Yaskawa INFORM job: A_ROOF_UPPER_0614_2_PAINT_15.JBI

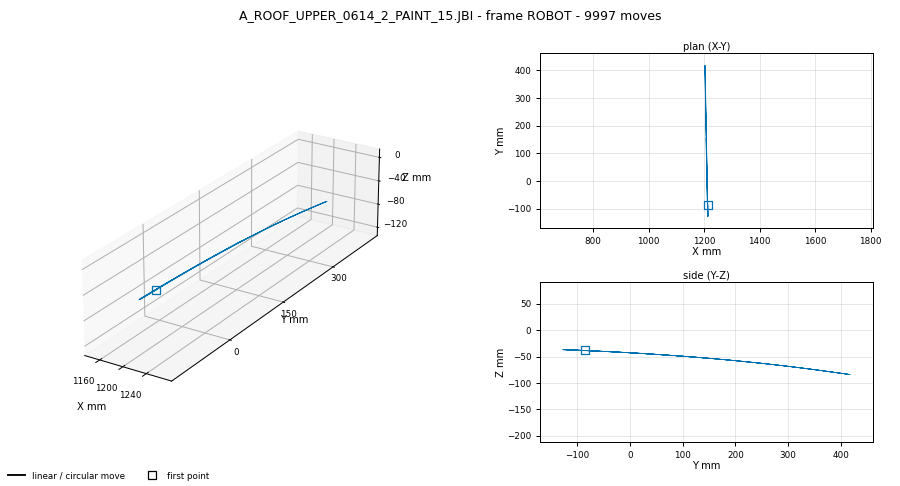
[picture p0: tool path of A_ROOF_UPPER_0614_2_PAINT_15.JBI in frame ROBOT, 9997 of 9997 moves have a stored position in this frame; points joined in program order, loops and branches not executed]
/JOB
//NAME A_ROOF_UPPER_0614_2_PAINT15
//POS
///NPOS 9997,0,0,0,0,0
///TOOL 1
///USER 0
///POSTYPE ROBOT
///RECTAN
///RCONF 1,0,0,0,0,0,0,0,0,0,0,0,0,0,0,0,0,0,0,0,0,0,0,0
C00000=1213.406,-85.221,-38.289,179.521,5.425,149.092
C00001=1213.411,-85.470,-38.278,179.518,5.424,149.093
C00002=1213.416,-85.720,-38.268,179.516,5.425,149.094
C00003=1213.422,-85.969,-38.257,179.513,5.424,149.094
C00004=1213.427,-86.220,-38.246,179.511,5.425,149.095
C00005=1213.432,-86.469,-38.234,179.509,5.424,149.095
C00006=1213.438,-86.719,-38.224,179.507,5.424,149.096
C00007=1213.443,-86.969,-38.213,179.504,5.424,149.097
C00008=1213.448,-87.218,-38.203,179.502,5.423,149.098
C00009=1213.453,-87.468,-38.192,179.500,5.424,149.098
C00010=1213.458,-87.717,-38.181,179.497,5.423,149.099
C00011=1213.463,-87.968,-38.170,179.495,5.424,149.100
C00012=1213.469,-88.217,-38.160,179.493,5.423,149.100
C00013=1213.474,-88.467,-38.149,179.491,5.423,149.101
C00014=1213.479,-88.717,-38.138,179.488,5.423,149.102
C00015=1213.484,-88.967,-38.128,179.486,5.423,149.102
C00016=1213.489,-89.216,-38.117,179.483,5.423,149.103
C00017=1213.495,-89.466,-38.107,179.481,5.423,149.104
C00018=1213.500,-89.716,-38.096,179.478,5.423,149.105
C00019=1213.506,-89.965,-38.085,179.477,5.423,149.105
C00020=1213.511,-90.215,-38.074,179.474,5.422,149.106
C00021=1213.516,-90.465,-38.064,179.472,5.423,149.106
C00022=1213.521,-90.715,-38.053,179.469,5.422,149.107
C00023=1213.526,-90.964,-38.042,179.467,5.423,149.108
C00024=1213.531,-91.214,-38.032,179.465,5.422,149.109
C00025=1213.537,-91.463,-38.021,179.463,5.422,149.109
C00026=1213.542,-91.714,-38.010,179.460,5.422,149.110
C00027=1213.547,-91.963,-38.000,179.458,5.421,149.110
C00028=1213.552,-92.213,-37.989,179.456,5.422,149.111
C00029=1213.558,-92.462,-37.979,179.453,5.421,149.112
C00030=1213.563,-92.713,-37.968,179.451,5.422,149.113
C00031=1213.568,-92.962,-37.958,179.449,5.421,149.113
C00032=1213.573,-93.212,-37.947,179.446,5.421,149.114
C00033=1213.578,-93.461,-37.936,179.444,5.421,149.114
C00034=1213.584,-93.711,-37.926,179.442,5.421,149.115
C00035=1213.589,-93.961,-37.915,179.439,5.421,149.116
C00036=1213.595,-94.211,-37.905,179.437,5.421,149.117
C00037=1213.599,-94.460,-37.894,179.435,5.420,149.117
C00038=1213.605,-94.710,-37.884,179.433,5.421,149.118
C00039=1213.610,-94.960,-37.873,179.430,5.420,149.119
C00040=1213.615,-95.209,-37.864,179.428,5.421,149.119
C00041=1213.620,-95.459,-37.853,179.425,5.420,149.120
C00042=1213.625,-95.709,-37.843,179.423,5.421,149.121
C00043=1213.631,-95.958,-37.832,179.421,5.420,149.121
C00044=1213.636,-96.208,-37.821,179.419,5.420,149.122
C00045=1213.641,-96.458,-37.811,179.416,5.420,149.123
C00046=1213.646,-96.708,-37.801,179.414,5.420,149.123
C00047=1213.652,-96.957,-37.790,179.411,5.420,149.124
C00048=1213.657,-97.208,-37.780,179.409,5.420,149.125
C00049=1213.662,-97.457,-37.770,179.407,5.419,149.125
C00050=1213.668,-97.706,-37.759,179.405,5.420,149.126
C00051=1213.673,-97.956,-37.748,179.402,5.419,149.127
C00052=1213.678,-98.206,-37.738,179.400,5.419,149.127
C00053=1213.683,-98.456,-37.728,179.398,5.419,149.128
C00054=1213.688,-98.705,-37.718,179.396,5.419,149.129
C00055=1213.694,-98.955,-37.707,179.393,5.419,149.129
C00056=1213.699,-99.205,-37.697,179.391,5.419,149.130
C00057=1213.704,-99.455,-37.687,179.389,5.419,149.131
C00058=1213.709,-99.705,-37.676,179.387,5.419,149.131
C00059=1213.715,-99.955,-37.666,179.384,5.419,149.132
C00060=1213.720,-100.204,-37.656,179.382,5.419,149.133
C00061=1213.725,-100.454,-37.646,179.380,5.418,149.133
C00062=1213.731,-100.725,-37.635,179.377,5.418,149.134
C00063=1213.737,-100.996,-37.624,179.375,5.418,149.135
C00064=1213.743,-101.268,-37.612,179.372,5.418,149.135
C00065=1213.747,-101.539,-37.600,179.370,5.418,149.136
C00066=1213.753,-101.788,-37.590,179.367,5.418,149.137
C00067=1213.759,-102.038,-37.580,179.365,5.418,149.138
C00068=1213.763,-102.288,-37.570,179.363,5.418,149.138
C00069=1213.768,-102.537,-37.560,179.360,5.418,149.139
C00070=1213.774,-102.787,-37.550,179.358,5.417,149.139
C00071=1213.779,-103.038,-37.540,179.356,5.417,149.140
C00072=1213.785,-103.287,-37.529,179.354,5.417,149.141
C00073=1213.790,-103.536,-37.520,179.351,5.417,149.142
C00074=1213.795,-103.787,-37.509,179.349,5.417,149.142
C00075=1213.800,-104.036,-37.499,179.347,5.417,149.143
C00076=1213.806,-104.286,-37.489,179.344,5.417,149.144
C00077=1213.810,-104.536,-37.479,179.342,5.417,149.144
C00078=1213.816,-104.785,-37.469,179.340,5.417,149.145
C00079=1213.821,-105.035,-37.458,179.338,5.417,149.146
C00080=1213.826,-105.285,-37.448,179.335,5.417,149.146
C00081=1213.831,-105.534,-37.438,179.333,5.416,149.147
C00082=1213.837,-105.784,-37.428,179.331,5.416,149.148
C00083=1213.842,-106.034,-37.418,179.329,5.416,149.148
C00084=1213.848,-106.284,-37.408,179.326,5.416,149.149
C00085=1213.853,-106.533,-37.398,179.324,5.416,149.150
C00086=1213.858,-106.784,-37.388,179.322,5.416,149.150
C00087=1213.863,-107.033,-37.378,179.320,5.416,149.151
C00088=1213.868,-107.282,-37.368,179.317,5.416,149.152
C00089=1213.874,-107.532,-37.358,179.315,5.416,149.152
C00090=1213.879,-107.782,-37.347,179.313,5.415,149.153
C00091=1213.885,-108.032,-37.338,179.311,5.416,149.154
C00092=1213.890,-108.281,-37.328,179.308,5.415,149.154
C00093=1213.895,-108.532,-37.318,179.306,5.415,149.155
C00094=1213.900,-108.781,-37.307,179.303,5.415,149.156
C00095=1213.905,-109.031,-37.298,179.301,5.415,149.156
C00096=1213.911,-109.280,-37.288,179.299,5.415,149.157
C00097=1213.916,-109.531,-37.278,179.297,5.415,149.158
C00098=1213.921,-109.780,-37.268,179.295,5.415,149.158
C00099=1213.926,-110.030,-37.258,179.292,5.415,149.159
C00100=1213.932,-110.279,-37.248,179.290,5.415,149.160
C00101=1213.936,-110.530,-37.238,179.288,5.415,149.160
C00102=1213.942,-110.779,-37.228,179.286,5.415,149.161
C00103=1213.947,-111.029,-37.219,179.283,5.415,149.162
C00104=1213.953,-111.278,-37.208,179.281,5.415,149.162
C00105=1213.958,-111.528,-37.198,179.279,5.414,149.163
C00106=1213.963,-111.778,-37.189,179.277,5.415,149.164
C00107=1213.968,-112.028,-37.179,179.274,5.414,149.164
C00108=1213.974,-112.277,-37.168,179.272,5.414,149.165
C00109=1213.979,-112.527,-37.160,179.270,5.414,149.166
C00110=1213.984,-112.777,-37.149,179.267,5.414,149.166
C00111=1213.989,-113.027,-37.139,179.265,5.414,149.167
C00112=1213.995,-113.276,-37.129,179.263,5.414,149.168
C00113=1214.000,-113.526,-37.120,179.260,5.413,149.168
C00114=1214.005,-113.776,-37.110,179.258,5.414,149.169
C00115=1214.010,-114.026,-37.099,179.256,5.413,149.170
C00116=1214.015,-114.276,-37.091,179.254,5.414,149.170
C00117=1214.021,-114.525,-37.080,179.251,5.413,149.171
C00118=1214.026,-114.774,-37.071,179.249,5.413,149.171
C00119=1214.032,-115.025,-37.061,179.247,5.414,149.172
C00120=1214.037,-115.275,-37.051,179.245,5.413,149.173
C00121=1214.042,-115.525,-37.042,179.243,5.413,149.173
C00122=1214.048,-115.774,-37.032,179.240,5.413,149.174
C00123=1214.052,-116.023,-37.022,179.238,5.413,149.175
C00124=1214.058,-116.274,-37.012,179.236,5.413,149.176
C00125=1214.063,-116.523,-37.003,179.233,5.413,149.176
C00126=1214.068,-116.773,-36.992,179.231,5.412,149.177
C00127=1214.073,-117.023,-36.983,179.229,5.413,149.177
C00128=1214.079,-117.272,-36.973,179.226,5.412,149.178
C00129=1214.084,-117.522,-36.964,179.224,5.413,149.179
C00130=1214.090,-117.772,-36.954,179.222,5.412,149.179
C00131=1214.095,-118.021,-36.944,179.220,5.412,149.180
C00132=1214.100,-118.272,-36.935,179.217,5.412,149.181
C00133=1214.105,-118.521,-36.925,179.215,5.412,149.182
C00134=1214.111,-118.771,-36.915,179.213,5.411,149.182
C00135=1214.116,-119.021,-36.906,179.211,5.412,149.183
C00136=1214.121,-119.271,-36.896,179.209,5.412,149.183
C00137=1214.126,-119.520,-36.887,179.206,5.412,149.184
C00138=1214.132,-119.770,-36.877,179.205,5.412,149.185
C00139=1214.137,-120.019,-36.868,179.202,5.411,149.185
C00140=1214.142,-120.270,-36.858,179.200,5.412,149.186
C00141=1214.147,-120.520,-36.848,179.198,5.411,149.187
C00142=1214.153,-120.770,-36.839,179.196,5.411,149.187
C00143=1214.158,-121.019,-36.829,179.193,5.411,149.188
C00144=1214.163,-121.269,-36.820,179.191,5.411,149.189
C00145=1214.169,-121.518,-36.810,179.189,5.411,149.189
C00146=1214.174,-121.768,-36.801,179.187,5.411,149.190
C00147=1214.180,-122.018,-36.791,179.184,5.411,149.191
C00148=1214.185,-122.268,-36.782,179.182,5.411,149.191
C00149=1214.190,-122.518,-36.771,179.180,5.411,149.192
C00150=1214.195,-122.768,-36.762,179.178,5.411,149.193
C00151=1214.200,-123.017,-36.753,179.175,5.411,149.193
C00152=1214.206,-123.267,-36.743,179.173,5.410,149.194
C00153=1214.211,-123.517,-36.734,179.171,5.410,149.194
C00154=1214.216,-123.766,-36.724,179.168,5.410,149.195
C00155=1214.222,-124.016,-36.715,179.166,5.410,149.196
C00156=1214.226,-124.265,-36.706,179.164,5.410,149.196
C00157=1214.232,-124.516,-36.696,179.162,5.410,149.197
C00158=1214.237,-124.765,-36.687,179.159,5.410,149.198
C00159=1214.242,-125.015,-36.678,179.157,5.410,149.199
C00160=1214.248,-125.265,-36.668,179.156,5.410,149.199
C00161=1214.253,-125.514,-36.659,179.153,5.410,149.200
C00162=1214.259,-125.764,-36.649,179.151,5.410,149.200
C00163=1214.264,-126.014,-36.640,179.148,5.410,149.201
C00164=1214.268,-126.264,-36.630,179.147,5.410,149.202
C00165=1214.274,-126.514,-36.621,179.144,5.409,149.202
C00166=1213.853,-126.525,-36.659,179.140,5.412,149.204
C00167=1213.848,-126.275,-36.668,179.142,5.413,149.204
C00168=1213.842,-126.025,-36.677,179.144,5.413,149.203
C00169=1213.837,-125.775,-36.687,179.147,5.413,149.202
C00170=1213.832,-125.526,-36.696,179.149,5.413,149.202
C00171=1213.826,-125.276,-36.705,179.151,5.414,149.201
C00172=1213.821,-125.026,-36.715,179.153,5.413,149.200
C00173=1213.816,-124.776,-36.724,179.155,5.413,149.200
C00174=1213.810,-124.527,-36.734,179.158,5.414,149.199
C00175=1213.805,-124.277,-36.743,179.160,5.413,149.198
C00176=1213.800,-124.027,-36.752,179.162,5.414,149.198
C00177=1213.794,-123.777,-36.762,179.165,5.413,149.197
C00178=1213.790,-123.527,-36.771,179.167,5.414,149.197
C00179=1213.785,-123.278,-36.781,179.169,5.414,149.196
C00180=1213.779,-123.028,-36.790,179.172,5.414,149.195
C00181=1213.774,-122.778,-36.799,179.173,5.414,149.195
C00182=1213.768,-122.528,-36.809,179.176,5.414,149.194
C00183=1213.763,-122.278,-36.818,179.178,5.414,149.193
C00184=1213.758,-122.029,-36.828,179.180,5.414,149.193
C00185=1213.752,-121.779,-36.837,179.182,5.414,149.192
C00186=1213.747,-121.530,-36.847,179.184,5.414,149.191
C00187=1213.741,-121.279,-36.857,179.187,5.415,149.191
C00188=1213.737,-121.030,-36.866,179.189,5.414,149.190
C00189=1213.731,-120.779,-36.876,179.191,5.415,149.189
C00190=1213.726,-120.530,-36.886,179.193,5.415,149.189
C00191=1213.720,-120.280,-36.895,179.196,5.415,149.188
C00192=1213.716,-120.031,-36.905,179.198,5.415,149.187
C00193=1213.710,-119.781,-36.914,179.200,5.415,149.187
C00194=1213.705,-119.531,-36.924,179.202,5.415,149.186
C00195=1213.700,-119.282,-36.933,179.205,5.415,149.185
C00196=1213.694,-119.032,-36.943,179.207,5.415,149.185
C00197=1213.689,-118.782,-36.952,179.209,5.415,149.184
C00198=1213.684,-118.532,-36.962,179.211,5.415,149.183
C00199=1213.679,-118.282,-36.971,179.213,5.415,149.183
C00200=1213.673,-118.032,-36.982,179.216,5.416,149.182
C00201=1213.668,-117.783,-36.991,179.218,5.415,149.181
C00202=1213.662,-117.533,-37.001,179.220,5.416,149.181
C00203=1213.658,-117.284,-37.010,179.223,5.415,149.180
C00204=1213.652,-117.033,-37.020,179.225,5.416,149.180
C00205=1213.647,-116.784,-37.030,179.227,5.416,149.179
C00206=1213.641,-116.534,-37.039,179.230,5.416,149.178
C00207=1213.637,-116.284,-37.049,179.232,5.416,149.177
C00208=1213.631,-116.035,-37.059,179.234,5.417,149.177
C00209=1213.626,-115.785,-37.068,179.236,5.416,149.176
C00210=1213.621,-115.535,-37.079,179.239,5.417,149.175
C00211=1213.616,-115.286,-37.088,179.241,5.416,149.175
C00212=1213.610,-115.035,-37.098,179.243,5.417,149.174
C00213=1213.604,-114.786,-37.108,179.245,5.417,149.174
C00214=1213.599,-114.536,-37.117,179.247,5.416,149.173
C00215=1213.594,-114.286,-37.127,179.250,5.417,149.172
C00216=1213.589,-114.036,-37.137,179.251,5.417,149.172
C00217=1213.584,-113.786,-37.146,179.254,5.417,149.171
C00218=1213.579,-113.537,-37.156,179.256,5.417,149.170
C00219=1213.573,-113.288,-37.166,179.259,5.417,149.170
C00220=1213.567,-113.037,-37.176,179.261,5.417,149.169
C00221=1213.563,-112.787,-37.186,179.263,5.418,149.168
C00222=1213.557,-112.538,-37.196,179.265,5.417,149.168
C00223=1213.552,-112.289,-37.206,179.268,5.418,149.167
C00224=1213.547,-112.038,-37.215,179.270,5.417,149.166
C00225=1213.541,-111.789,-37.225,179.272,5.418,149.166
C00226=1213.537,-111.539,-37.235,179.274,5.418,149.165
C00227=1213.531,-111.289,-37.245,179.277,5.418,149.164
C00228=1213.525,-111.039,-37.255,179.279,5.418,149.164
C00229=1213.520,-110.790,-37.265,179.281,5.419,149.163
C00230=1213.515,-110.540,-37.275,179.283,5.418,149.162
C00231=1213.510,-110.291,-37.285,179.286,5.419,149.162
C00232=1213.505,-110.040,-37.294,179.288,5.418,149.161
C00233=1213.499,-109.791,-37.304,179.291,5.419,149.160
C00234=1213.495,-109.541,-37.314,179.292,5.419,149.160
C00235=1213.489,-109.291,-37.325,179.294,5.418,149.159
C00236=1213.483,-109.041,-37.334,179.297,5.419,149.158
C00237=1213.478,-108.792,-37.344,179.299,5.418,149.158
C00238=1213.473,-108.542,-37.354,179.302,5.419,149.157
C00239=1213.468,-108.292,-37.364,179.303,5.419,149.156
C00240=1213.463,-108.043,-37.374,179.306,5.419,149.156
C00241=1213.457,-107.793,-37.384,179.308,5.419,149.155
C00242=1213.452,-107.543,-37.394,179.311,5.419,149.154
C00243=1213.446,-107.293,-37.404,179.312,5.419,149.154
C00244=1213.442,-107.044,-37.414,179.315,5.420,149.153
C00245=1213.437,-106.794,-37.425,179.317,5.419,149.152
C00246=1213.431,-106.544,-37.435,179.320,5.420,149.152
C00247=1213.426,-106.295,-37.444,179.322,5.419,149.151
C00248=1213.420,-106.045,-37.455,179.324,5.420,149.150
C00249=1213.415,-105.794,-37.464,179.326,5.420,149.150
C00250=1213.410,-105.545,-37.475,179.329,5.420,149.149
C00251=1213.405,-105.296,-37.484,179.331,5.420,149.148
C00252=1213.400,-105.045,-37.495,179.334,5.420,149.148
C00253=1213.394,-104.796,-37.505,179.335,5.420,149.147
C00254=1213.389,-104.546,-37.515,179.338,5.420,149.146
C00255=1213.384,-104.296,-37.525,179.340,5.420,149.146
C00256=1213.379,-104.047,-37.535,179.343,5.421,149.145
C00257=1213.373,-103.797,-37.546,179.345,5.420,149.144
C00258=1213.368,-103.547,-37.556,179.347,5.421,149.144
C00259=1213.363,-103.298,-37.566,179.349,5.421,149.143
C00260=1213.358,-103.048,-37.576,179.352,5.421,149.142
C00261=1213.353,-102.798,-37.587,179.354,5.421,149.142
C00262=1213.347,-102.548,-37.597,179.357,5.421,149.141
C00263=1213.342,-102.299,-37.606,179.358,5.421,149.140
C00264=1213.337,-102.049,-37.617,179.361,5.421,149.140
C00265=1213.332,-101.799,-37.627,179.363,5.421,149.139
C00266=1213.326,-101.550,-37.637,179.366,5.422,149.138
C00267=1213.321,-101.279,-37.648,179.368,5.421,149.138
C00268=1213.315,-101.007,-37.660,179.370,5.422,149.137
C00269=1213.310,-100.736,-37.671,179.373,5.422,149.136
C00270=1213.303,-100.465,-37.682,179.375,5.422,149.135
C00271=1213.299,-100.215,-37.692,179.378,5.422,149.135
C00272=1213.293,-99.965,-37.702,179.380,5.422,149.134
C00273=1213.288,-99.716,-37.712,179.382,5.422,149.133
C00274=1213.283,-99.466,-37.723,179.384,5.422,149.133
C00275=1213.277,-99.216,-37.733,179.387,5.423,149.132
C00276=1213.272,-98.966,-37.744,179.389,5.422,149.131
C00277=1213.266,-98.716,-37.754,179.392,5.423,149.131
C00278=1213.262,-98.467,-37.764,179.393,5.423,149.130
C00279=1213.257,-98.217,-37.774,179.396,5.423,149.129
C00280=1213.251,-97.967,-37.784,179.398,5.423,149.129
C00281=1213.246,-97.717,-37.795,179.401,5.423,149.128
C00282=1213.241,-97.468,-37.806,179.403,5.423,149.127
C00283=1213.235,-97.218,-37.816,179.405,5.423,149.127
C00284=1213.230,-96.968,-37.827,179.407,5.423,149.126
C00285=1213.225,-96.719,-37.837,179.410,5.424,149.125
C00286=1213.220,-96.468,-37.847,179.412,5.423,149.125
C00287=1213.214,-96.219,-37.858,179.414,5.424,149.124
C00288=1213.210,-95.969,-37.868,179.417,5.423,149.123
C00289=1213.204,-95.719,-37.878,179.419,5.424,149.123
C00290=1213.199,-95.470,-37.889,179.421,5.424,149.122
C00291=1213.194,-95.220,-37.899,179.423,5.424,149.121
C00292=1213.188,-94.971,-37.910,179.426,5.424,149.121
C00293=1213.183,-94.720,-37.920,179.428,5.424,149.120
C00294=1213.178,-94.471,-37.930,179.430,5.424,149.119
C00295=1213.173,-94.221,-37.942,179.433,5.425,149.119
C00296=1213.167,-93.972,-37.952,179.435,5.424,149.118
C00297=1213.162,-93.721,-37.962,179.437,5.425,149.117
C00298=1213.157,-93.472,-37.973,179.439,5.424,149.117
C00299=1213.151,-93.222,-37.983,179.442,5.425,149.116
C00300=1213.146,-92.973,-37.994,179.444,5.424,149.115
C00301=1213.141,-92.723,-38.004,179.446,5.425,149.115
C00302=1213.136,-92.473,-38.015,179.449,5.426,149.114
C00303=1213.130,-92.223,-38.025,179.451,5.425,149.113
C00304=1213.126,-91.974,-38.036,179.454,5.426,149.113
C00305=1213.120,-91.724,-38.047,179.456,5.425,149.112
C00306=1213.115,-91.474,-38.057,179.459,5.426,149.111
C00307=1213.109,-91.224,-38.067,179.460,5.426,149.111
C00308=1213.105,-90.975,-38.079,179.463,5.426,149.110
C00309=1213.099,-90.725,-38.089,179.465,5.426,149.109
C00310=1213.094,-90.475,-38.099,179.468,5.426,149.109
C00311=1213.089,-90.226,-38.110,179.470,5.426,149.108
C00312=1213.084,-89.976,-38.121,179.472,5.426,149.107
C00313=1213.078,-89.726,-38.131,179.474,5.426,149.106
C00314=1213.073,-89.477,-38.142,179.477,5.427,149.106
C00315=1213.068,-89.227,-38.153,179.479,5.426,149.105
C00316=1213.063,-88.977,-38.163,179.481,5.427,149.104
C00317=1213.058,-88.728,-38.174,179.483,5.426,149.104
C00318=1213.053,-88.478,-38.185,179.486,5.427,149.103
C00319=1213.047,-88.228,-38.195,179.488,5.426,149.102
C00320=1213.042,-87.978,-38.207,179.490,5.427,149.102
C00321=1213.037,-87.728,-38.217,179.492,5.427,149.101
C00322=1213.031,-87.479,-38.228,179.495,5.427,149.100
C00323=1213.026,-87.229,-38.239,179.498,5.428,149.100
C00324=1213.021,-86.979,-38.249,179.500,5.427,149.099
C00325=1213.016,-86.730,-38.260,179.503,5.428,149.098
C00326=1213.010,-86.480,-38.271,179.505,5.427,149.098
C00327=1213.005,-86.230,-38.281,179.507,5.428,149.097
C00328=1213.000,-85.981,-38.292,179.509,5.428,149.096
C00329=1212.995,-85.731,-38.303,179.512,5.428,149.096
C00330=1212.990,-85.481,-38.315,179.514,5.428,149.095
C00331=1212.984,-85.231,-38.325,179.516,5.428,149.094
C00332=1212.979,-84.982,-38.336,179.518,5.428,149.094
C00333=1212.974,-84.732,-38.346,179.521,5.428,149.093
C00334=1212.969,-84.483,-38.358,179.523,5.429,149.092
C00335=1212.964,-84.232,-38.368,179.525,5.429,149.092
C00336=1212.959,-83.983,-38.379,179.527,5.429,149.091
C00337=1212.953,-83.733,-38.390,179.530,5.429,149.090
C00338=1212.947,-83.483,-38.400,179.533,5.429,149.090
C00339=1212.943,-83.234,-38.412,179.535,5.429,149.089
C00340=1212.938,-82.983,-38.422,179.538,5.430,149.088
C00341=1212.932,-82.734,-38.433,179.539,5.430,149.088
C00342=1212.928,-82.485,-38.445,179.542,5.430,149.087
C00343=1212.921,-82.235,-38.455,179.544,5.430,149.086
C00344=1212.917,-81.985,-38.467,179.547,5.430,149.086
C00345=1212.912,-81.735,-38.477,179.549,5.430,149.085
C00346=1212.906,-81.486,-38.488,179.551,5.430,149.084
C00347=1212.901,-81.236,-38.499,179.553,5.430,149.083
C00348=1212.895,-80.987,-38.510,179.556,5.431,149.083
C00349=1212.890,-80.736,-38.521,179.558,5.431,149.082
C00350=1212.886,-80.487,-38.532,179.560,5.431,149.081
C00351=1212.880,-80.238,-38.543,179.563,5.431,149.081
C00352=1212.875,-79.988,-38.554,179.565,5.431,149.080
C00353=1212.870,-79.738,-38.565,179.568,5.431,149.079
C00354=1212.864,-79.488,-38.576,179.570,5.431,149.079
C00355=1212.860,-79.239,-38.587,179.572,5.432,149.078
C00356=1212.855,-78.989,-38.598,179.574,5.431,149.077
C00357=1212.849,-78.739,-38.609,179.577,5.432,149.077
C00358=1212.844,-78.489,-38.620,179.579,5.431,149.076
C00359=1212.839,-78.239,-38.631,179.582,5.432,149.075
C00360=1212.833,-77.990,-38.642,179.584,5.432,149.075
C00361=1212.828,-77.740,-38.654,179.586,5.432,149.074
C00362=1212.823,-77.490,-38.664,179.589,5.432,149.073
C00363=1212.818,-77.241,-38.675,179.591,5.432,149.073
C00364=1212.813,-76.991,-38.687,179.593,5.433,149.072
C00365=1212.808,-76.741,-38.698,179.595,5.432,149.071
C00366=1212.802,-76.492,-38.709,179.598,5.433,149.071
C00367=1212.797,-76.242,-38.721,179.600,5.432,149.070
C00368=1212.792,-75.992,-38.731,179.603,5.433,149.069
C00369=1212.787,-75.743,-38.742,179.606,5.433,149.068
C00370=1212.781,-75.493,-38.754,179.608,5.433,149.068
C00371=1212.776,-75.222,-38.766,179.610,5.433,149.067
C00372=1212.770,-74.952,-38.777,179.613,5.434,149.066
C00373=1212.764,-74.681,-38.790,179.615,5.434,149.066
C00374=1212.759,-74.411,-38.803,179.618,5.434,149.065
C00375=1212.754,-74.161,-38.813,179.620,5.434,149.064
C00376=1212.748,-73.911,-38.825,179.622,5.434,149.064
C00377=1212.743,-73.662,-38.836,179.625,5.435,149.063
C00378=1212.739,-73.412,-38.847,179.627,5.434,149.062
C00379=1212.732,-73.162,-38.858,179.629,5.435,149.062
C00380=1212.728,-72.913,-38.869,179.631,5.435,149.061
C00381=1212.722,-72.663,-38.881,179.634,5.435,149.060
C00382=1212.717,-72.414,-38.892,179.636,5.435,149.059
C00383=1212.712,-72.164,-38.904,179.639,5.435,149.059
C00384=1212.707,-71.913,-38.915,179.642,5.436,149.058
C00385=1212.702,-71.664,-38.926,179.644,5.435,149.057
C00386=1212.696,-71.415,-38.937,179.646,5.436,149.057
C00387=1212.691,-71.165,-38.949,179.648,5.436,149.056
C00388=1212.686,-70.915,-38.960,179.651,5.436,149.055
C00389=1212.681,-70.665,-38.972,179.653,5.436,149.055
C00390=1212.675,-70.416,-38.982,179.655,5.436,149.054
C00391=1212.670,-70.166,-38.994,179.658,5.437,149.053
C00392=1212.665,-69.916,-39.005,179.660,5.436,149.053
C00393=1212.660,-69.666,-39.017,179.663,5.437,149.052
C00394=1212.655,-69.417,-39.029,179.665,5.436,149.051
C00395=1212.649,-69.168,-39.040,179.668,5.437,149.051
C00396=1212.644,-68.918,-39.051,179.669,5.437,149.050
C00397=1212.639,-68.668,-39.063,179.672,5.437,149.049
C00398=1212.634,-68.418,-39.075,179.674,5.438,149.049
C00399=1212.629,-68.168,-39.085,179.677,5.437,149.048
C00400=1212.623,-67.919,-39.097,179.679,5.438,149.047
C00401=1212.619,-67.669,-39.108,179.681,5.438,149.047
C00402=1212.613,-67.419,-39.120,179.684,5.438,149.046
C00403=1212.608,-67.170,-39.131,179.687,5.438,149.045
C00404=1212.603,-66.920,-39.143,179.689,5.438,149.044
C00405=1212.598,-66.671,-39.154,179.691,5.439,149.044
C00406=1212.592,-66.421,-39.166,179.693,5.439,149.043
C00407=1212.588,-66.171,-39.177,179.696,5.439,149.042
C00408=1212.582,-65.921,-39.189,179.698,5.439,149.042
C00409=1212.577,-65.671,-39.201,179.700,5.439,149.041
C00410=1212.572,-65.422,-39.212,179.703,5.440,149.040
C00411=1212.566,-65.173,-39.224,179.705,5.439,149.040
C00412=1212.561,-64.923,-39.235,179.708,5.440,149.039
C00413=1212.556,-64.673,-39.247,179.710,5.439,149.038
C00414=1212.551,-64.423,-39.258,179.712,5.440,149.038
C00415=1212.546,-64.173,-39.270,179.715,5.441,149.037
C00416=1212.541,-63.924,-39.281,179.717,5.440,149.036
C00417=1212.536,-63.674,-39.293,179.720,5.441,149.036
C00418=1212.530,-63.425,-39.304,179.722,5.440,149.035
C00419=1212.525,-63.175,-39.316,179.724,5.441,149.034
C00420=1212.520,-62.925,-39.328,179.727,5.441,149.034
C00421=1212.515,-62.675,-39.339,179.729,5.441,149.033
C00422=1212.510,-62.426,-39.352,179.732,5.441,149.032
C00423=1212.505,-62.176,-39.363,179.734,5.441,149.031
C00424=1212.500,-61.927,-39.375,179.736,5.442,149.031
C00425=1212.494,-61.677,-39.387,179.739,5.442,149.030
C00426=1212.489,-61.427,-39.398,179.741,5.442,149.030
C00427=1212.483,-61.178,-39.410,179.743,5.442,149.029
C00428=1212.479,-60.928,-39.421,179.745,5.442,149.028
C00429=1212.473,-60.678,-39.433,179.748,5.442,149.027
C00430=1212.468,-60.429,-39.445,179.751,5.443,149.027
C00431=1212.464,-60.179,-39.457,179.753,5.443,149.026
C00432=1212.458,-59.929,-39.469,179.756,5.443,149.025
C00433=1212.453,-59.679,-39.480,179.758,5.443,149.025
C00434=1212.448,-59.430,-39.492,179.760,5.444,149.024
C00435=1212.443,-59.180,-39.504,179.763,5.444,149.023
C00436=1212.437,-58.930,-39.516,179.765,5.444,149.023
C00437=1212.433,-58.681,-39.528,179.767,5.444,149.022
C00438=1212.427,-58.431,-39.539,179.769,5.444,149.021
C00439=1212.422,-58.181,-39.551,179.772,5.444,149.021
C00440=1212.417,-57.932,-39.562,179.775,5.445,149.020
C00441=1212.411,-57.683,-39.575,179.777,5.444,149.019
C00442=1212.406,-57.433,-39.587,179.779,5.445,149.018
C00443=1212.401,-57.183,-39.598,179.782,5.444,149.018
C00444=1212.396,-56.933,-39.610,179.784,5.445,149.017
C00445=1212.391,-56.684,-39.622,179.786,5.446,149.017
C00446=1212.386,-56.434,-39.634,179.788,5.445,149.016
C00447=1212.381,-56.184,-39.646,179.791,5.446,149.015
C00448=1212.375,-55.934,-39.658,179.793,5.445,149.014
C00449=1212.370,-55.685,-39.670,179.796,5.446,149.014
C00450=1212.365,-55.435,-39.681,179.799,5.446,149.013
C00451=1212.360,-55.186,-39.693,179.801,5.446,149.012
C00452=1212.355,-54.936,-39.706,179.803,5.447,149.012
C00453=1212.349,-54.686,-39.718,179.806,5.447,149.011
C00454=1212.345,-54.437,-39.729,179.808,5.447,149.010
C00455=1212.339,-54.187,-39.741,179.810,5.447,149.010
C00456=1212.334,-53.937,-39.754,179.812,5.447,149.009
C00457=1212.329,-53.687,-39.765,179.815,5.448,149.008
C00458=1212.324,-53.438,-39.777,179.818,5.448,149.008
C00459=1212.319,-53.189,-39.789,179.820,5.448,149.007
C00460=1212.314,-52.939,-39.801,179.822,5.448,149.006
C00461=1212.308,-52.689,-39.814,179.825,5.449,149.006
C00462=1212.304,-52.440,-39.825,179.827,5.448,149.005
C00463=1212.298,-52.190,-39.837,179.830,5.449,149.004
C00464=1212.293,-51.940,-39.850,179.832,5.448,149.003
C00465=1212.288,-51.690,-39.861,179.835,5.449,149.003
C00466=1212.283,-51.441,-39.874,179.837,5.450,149.002
C00467=1212.277,-51.191,-39.886,179.839,5.449,149.002
C00468=1212.272,-50.942,-39.897,179.841,5.450,149.001
C00469=1212.267,-50.692,-39.910,179.844,5.450,149.000
C00470=1212.262,-50.442,-39.922,179.846,5.450,148.999
C00471=1212.257,-50.192,-39.935,179.849,5.450,148.999
C00472=1212.252,-49.942,-39.947,179.851,5.450,148.998
C00473=1212.247,-49.693,-39.959,179.854,5.451,148.997
C00474=1212.242,-49.443,-39.970,179.856,5.451,148.997
C00475=1212.235,-49.173,-39.984,179.858,5.451,148.996
C00476=1212.230,-48.904,-39.997,179.861,5.451,148.995
C00477=1212.225,-48.633,-40.010,179.864,5.452,148.995
C00478=1212.219,-48.364,-40.023,179.866,5.452,148.994
C00479=1212.214,-48.114,-40.036,179.868,5.452,148.993
C00480=1212.209,-47.864,-40.047,179.871,5.452,148.992
C00481=1212.204,-47.614,-40.060,179.874,5.453,148.992
C00482=1212.199,-47.365,-40.072,179.876,5.452,148.991
C00483=1212.194,-47.115,-40.085,179.879,5.453,148.990
C00484=1212.188,-46.865,-40.097,179.881,5.453,148.990
C00485=1212.183,-46.616,-40.109,179.883,5.453,148.989
C00486=1212.178,-46.366,-40.121,179.886,5.453,148.988
C00487=1212.173,-46.117,-40.133,179.889,5.454,148.988
C00488=1212.168,-45.868,-40.146,179.890,5.454,148.987
C00489=1212.163,-45.618,-40.158,179.893,5.454,148.986
C00490=1212.158,-45.368,-40.170,179.896,5.455,148.986
C00491=1212.153,-45.118,-40.183,179.898,5.454,148.985
C00492=1212.148,-44.868,-40.195,179.900,5.455,148.984
C00493=1212.142,-44.619,-40.207,179.902,5.455,148.984
C00494=1212.137,-44.369,-40.220,179.905,5.455,148.983
C00495=1212.132,-44.120,-40.232,179.908,5.456,148.982
C00496=1212.127,-43.870,-40.244,179.910,5.455,148.981
C00497=1212.121,-43.621,-40.257,179.912,5.456,148.981
C00498=1212.116,-43.371,-40.269,179.915,5.456,148.980
C00499=1212.111,-43.121,-40.282,179.917,5.456,148.979
C00500=1212.106,-42.871,-40.294,179.919,5.457,148.979
C00501=1212.101,-42.622,-40.307,179.922,5.457,148.978
C00502=1212.096,-42.372,-40.319,179.924,5.457,148.977
C00503=1212.091,-42.123,-40.331,179.927,5.457,148.977
C00504=1212.086,-41.873,-40.344,179.929,5.458,148.976
C00505=1212.081,-41.623,-40.356,179.932,5.457,148.975
C00506=1212.076,-41.374,-40.369,179.934,5.458,148.975
C00507=1212.070,-41.124,-40.381,179.937,5.458,148.974
C00508=1212.065,-40.874,-40.393,179.939,5.458,148.973
C00509=1212.060,-40.625,-40.406,179.942,5.458,148.973
C00510=1212.055,-40.375,-40.419,179.944,5.459,148.972
C00511=1212.050,-40.126,-40.431,179.946,5.459,148.971
C00512=1212.045,-39.876,-40.443,179.949,5.459,148.971
C00513=1212.040,-39.626,-40.456,179.951,5.460,148.970
C00514=1212.034,-39.377,-40.469,179.953,5.460,148.969
C00515=1212.029,-39.127,-40.482,179.956,5.460,148.969
C00516=1212.024,-38.877,-40.494,179.959,5.461,148.968
C00517=1212.019,-38.627,-40.507,179.961,5.460,148.967
C00518=1212.014,-38.378,-40.519,179.963,5.461,148.966
C00519=1212.009,-38.129,-40.532,179.966,5.461,148.966
C00520=1212.004,-37.878,-40.544,179.968,5.461,148.965
C00521=1211.999,-37.629,-40.557,179.971,5.461,148.964
C00522=1211.993,-37.380,-40.569,179.973,5.462,148.964
C00523=1211.988,-37.130,-40.582,179.975,5.461,148.963
C00524=1211.982,-36.881,-40.595,179.978,5.462,148.963
C00525=1211.978,-36.631,-40.608,179.980,5.463,148.962
C00526=1211.973,-36.381,-40.620,179.982,5.462,148.961
C00527=1211.967,-36.131,-40.632,179.985,5.463,148.960
C00528=1211.962,-35.882,-40.645,179.988,5.463,148.960
C00529=1211.958,-35.632,-40.658,179.990,5.463,148.959
C00530=1211.953,-35.383,-40.671,179.992,5.463,148.958
C00531=1211.947,-35.133,-40.684,179.995,5.464,148.958
C00532=1211.942,-34.884,-40.696,179.998,5.464,148.957
C00533=1211.937,-34.634,-40.709,180.000,5.464,148.956
C00534=1211.932,-34.384,-40.721,-179.997,5.465,148.956
C00535=1211.927,-34.134,-40.734,-179.995,5.465,148.955
C00536=1211.921,-33.884,-40.747,-179.993,5.465,148.954
C00537=1211.916,-33.635,-40.760,-179.991,5.466,148.954
C00538=1211.911,-33.385,-40.773,-179.988,5.466,148.953
C00539=1211.906,-33.136,-40.785,-179.986,5.466,148.952
C00540=1211.901,-32.886,-40.798,-179.983,5.466,148.952
C00541=1211.896,-32.637,-40.811,-179.980,5.467,148.951
C00542=1211.890,-32.387,-40.824,-179.978,5.466,148.950
C00543=1211.886,-32.137,-40.837,-179.976,5.467,148.949
C00544=1211.881,-31.888,-40.850,-179.973,5.467,148.949
C00545=1211.875,-31.638,-40.863,-179.971,5.467,148.948
C00546=1211.870,-31.389,-40.875,-179.968,5.467,148.947
C00547=1211.865,-31.139,-40.888,-179.966,5.468,148.947
C00548=1211.860,-30.890,-40.901,-179.963,5.468,148.946
C00549=1211.854,-30.640,-40.914,-179.961,5.468,148.946
C00550=1211.850,-30.390,-40.927,-179.959,5.469,148.945
C00551=1211.845,-30.141,-40.940,-179.956,5.469,148.944
C00552=1211.840,-29.891,-40.952,-179.954,5.469,148.943
C00553=1211.834,-29.641,-40.966,-179.951,5.470,148.943
C00554=1211.829,-29.392,-40.978,-179.949,5.470,148.942
C00555=1211.824,-29.142,-40.991,-179.947,5.470,148.941
C00556=1211.819,-28.892,-41.004,-179.944,5.470,148.941
C00557=1211.814,-28.643,-41.017,-179.941,5.471,148.940
C00558=1211.809,-28.393,-41.030,-179.939,5.471,148.939
C00559=1211.804,-28.144,-41.043,-179.937,5.471,148.939
C00560=1211.798,-27.894,-41.057,-179.934,5.471,148.938
C00561=1211.794,-27.644,-41.070,-179.932,5.472,148.937
C00562=1211.789,-27.395,-41.082,-179.930,5.472,148.937
C00563=1211.783,-27.145,-41.095,-179.927,5.472,148.936
C00564=1211.778,-26.895,-41.108,-179.924,5.473,148.935
C00565=1211.773,-26.646,-41.121,-179.922,5.473,148.935
C00566=1211.768,-26.396,-41.135,-179.920,5.473,148.934
C00567=1211.763,-26.147,-41.148,-179.917,5.473,148.933
C00568=1211.758,-25.898,-41.160,-179.914,5.474,148.932
C00569=1211.753,-25.647,-41.174,-179.912,5.474,148.932
C00570=1211.748,-25.398,-41.187,-179.910,5.474,148.931
C00571=1211.742,-25.148,-41.200,-179.907,5.475,148.930
C00572=1211.737,-24.898,-41.213,-179.904,5.475,148.930
C00573=1211.732,-24.650,-41.226,-179.902,5.475,148.929
C00574=1211.727,-24.399,-41.240,-179.900,5.476,148.929
C00575=1211.722,-24.150,-41.252,-179.897,5.476,148.928
C00576=1211.718,-23.900,-41.265,-179.895,5.476,148.927
C00577=1211.712,-23.650,-41.278,-179.893,5.476,148.926
C00578=1211.707,-23.402,-41.292,-179.890,5.477,148.926
C00579=1211.701,-23.132,-41.306,-179.887,5.477,148.925
C00580=1211.696,-22.862,-41.321,-179.885,5.478,148.924
C00581=1211.691,-22.593,-41.335,-179.882,5.477,148.923
C00582=1211.684,-22.323,-41.349,-179.879,5.477,148.923
C00583=1211.680,-22.074,-41.362,-179.877,5.478,148.922
C00584=1211.674,-21.824,-41.376,-179.874,5.478,148.921
C00585=1211.670,-21.574,-41.388,-179.872,5.479,148.921
C00586=1211.664,-21.325,-41.402,-179.870,5.479,148.920
C00587=1211.660,-21.075,-41.415,-179.867,5.479,148.919
C00588=1211.654,-20.825,-41.429,-179.864,5.480,148.919
C00589=1211.650,-20.576,-41.442,-179.862,5.480,148.918
C00590=1211.644,-20.326,-41.455,-179.860,5.480,148.917
C00591=1211.639,-20.077,-41.468,-179.857,5.481,148.917
C00592=1211.634,-19.827,-41.482,-179.854,5.481,148.916
C00593=1211.629,-19.578,-41.495,-179.852,5.481,148.915
C00594=1211.623,-19.328,-41.508,-179.850,5.481,148.915
C00595=1211.618,-19.079,-41.522,-179.847,5.482,148.914
C00596=1211.613,-18.829,-41.535,-179.844,5.482,148.913
C00597=1211.608,-18.579,-41.548,-179.843,5.482,148.913
C00598=1211.603,-18.330,-41.562,-179.840,5.483,148.912
C00599=1211.598,-18.080,-41.575,-179.837,5.483,148.911
C00600=1211.593,-17.831,-41.589,-179.835,5.484,148.911
C00601=1211.588,-17.581,-41.602,-179.833,5.483,148.910
C00602=1211.583,-17.331,-41.615,-179.830,5.484,148.909
C00603=1211.578,-17.082,-41.629,-179.827,5.484,148.909
C00604=1211.573,-16.832,-41.642,-179.825,5.485,148.908
C00605=1211.568,-16.583,-41.655,-179.823,5.485,148.907
C00606=1211.562,-16.333,-41.669,-179.820,5.485,148.907
C00607=1211.557,-16.084,-41.683,-179.817,5.486,148.906
C00608=1211.552,-15.834,-41.696,-179.815,5.486,148.905
C00609=1211.547,-15.584,-41.710,-179.813,5.486,148.905
C00610=1211.542,-15.335,-41.723,-179.810,5.487,148.904
C00611=1211.537,-15.085,-41.737,-179.808,5.487,148.903
C00612=1211.532,-14.836,-41.750,-179.805,5.488,148.903
C00613=1211.527,-14.586,-41.764,-179.803,5.487,148.902
C00614=1211.521,-14.337,-41.777,-179.800,5.488,148.901
C00615=1211.517,-14.087,-41.791,-179.798,5.488,148.901
C00616=1211.511,-13.838,-41.804,-179.795,5.489,148.900
C00617=1211.506,-13.588,-41.818,-179.793,5.488,148.899
C00618=1211.502,-13.338,-41.831,-179.790,5.489,148.898
C00619=1211.496,-13.089,-41.845,-179.788,5.489,148.898
C00620=1211.491,-12.838,-41.859,-179.786,5.490,148.897
C00621=1211.486,-12.590,-41.872,-179.783,5.491,148.897
C00622=1211.481,-12.339,-41.886,-179.781,5.491,148.896
C00623=1211.476,-12.090,-41.900,-179.778,5.491,148.895
C00624=1211.471,-11.841,-41.913,-179.775,5.492,148.895
C00625=1211.466,-11.591,-41.927,-179.773,5.492,148.894
C00626=1211.460,-11.342,-41.941,-179.771,5.492,148.893
C00627=1211.456,-11.092,-41.954,-179.768,5.492,148.892
C00628=1211.451,-10.842,-41.968,-179.765,5.493,148.892
C00629=1211.445,-10.593,-41.982,-179.763,5.493,148.891
C00630=1211.441,-10.343,-41.995,-179.761,5.493,148.890
C00631=1211.435,-10.094,-42.009,-179.759,5.494,148.890
C00632=1211.430,-9.844,-42.023,-179.756,5.494,148.889
C00633=1211.426,-9.594,-42.036,-179.753,5.495,148.889
C00634=1211.420,-9.345,-42.050,-179.751,5.495,148.888
C00635=1211.415,-9.096,-42.064,-179.748,5.495,148.887
C00636=1211.410,-8.845,-42.078,-179.746,5.495,148.886
C00637=1211.405,-8.596,-42.091,-179.743,5.496,148.886
C00638=1211.400,-8.347,-42.105,-179.741,5.496,148.885
C00639=1211.395,-8.096,-42.119,-179.738,5.496,148.884
C00640=1211.389,-7.847,-42.133,-179.736,5.497,148.884
C00641=1211.385,-7.598,-42.146,-179.733,5.497,148.883
C00642=1211.380,-7.349,-42.160,-179.731,5.498,148.883
C00643=1211.374,-7.099,-42.174,-179.728,5.498,148.882
C00644=1211.369,-6.849,-42.188,-179.726,5.498,148.881
C00645=1211.365,-6.600,-42.202,-179.724,5.499,148.880
C00646=1211.360,-6.351,-42.216,-179.721,5.499,148.880
C00647=1211.354,-6.100,-42.229,-179.718,5.500,148.879
C00648=1211.349,-5.851,-42.244,-179.716,5.500,148.878
C00649=1211.344,-5.602,-42.258,-179.714,5.500,148.878
C00650=1211.340,-5.352,-42.271,-179.711,5.500,148.877
C00651=1211.335,-5.102,-42.285,-179.708,5.501,148.876
C00652=1211.329,-4.853,-42.299,-179.706,5.502,148.876
C00653=1211.324,-4.603,-42.313,-179.703,5.502,148.875
C00654=1211.319,-4.353,-42.327,-179.701,5.502,148.874
C00655=1211.313,-4.104,-42.341,-179.699,5.502,148.874
C00656=1211.309,-3.855,-42.355,-179.696,5.503,148.873
C00657=1211.304,-3.605,-42.369,-179.693,5.503,148.872
C00658=1211.299,-3.355,-42.383,-179.691,5.504,148.872
C00659=1211.293,-3.106,-42.397,-179.689,5.504,148.871
C00660=1211.288,-2.856,-42.411,-179.686,5.504,148.870
C00661=1211.284,-2.606,-42.425,-179.683,5.505,148.870
C00662=1211.278,-2.357,-42.439,-179.681,5.505,148.869
C00663=1211.274,-2.108,-42.453,-179.679,5.506,148.868
C00664=1211.269,-1.858,-42.467,-179.676,5.506,148.868
C00665=1211.264,-1.609,-42.481,-179.674,5.506,148.867
C00666=1211.258,-1.360,-42.495,-179.671,5.507,148.866
C00667=1211.253,-1.109,-42.509,-179.668,5.507,148.866
C00668=1211.248,-0.860,-42.523,-179.666,5.508,148.865
C00669=1211.243,-0.610,-42.537,-179.664,5.507,148.864
C00670=1211.238,-0.361,-42.551,-179.661,5.508,148.864
C00671=1211.233,-0.111,-42.566,-179.658,5.508,148.863
C00672=1211.228,0.139,-42.580,-179.656,5.509,148.862
C00673=1211.223,0.388,-42.594,-179.654,5.510,148.862
C00674=1211.218,0.638,-42.608,-179.651,5.510,148.861
C00675=1211.212,0.887,-42.622,-179.649,5.510,148.860
C00676=1211.208,1.136,-42.636,-179.646,5.510,148.860
C00677=1211.203,1.386,-42.650,-179.644,5.511,148.859
C00678=1211.198,1.636,-42.664,-179.641,5.511,148.858
C00679=1211.193,1.885,-42.678,-179.638,5.512,148.858
C00680=1211.188,2.135,-42.693,-179.636,5.512,148.857
C00681=1211.183,2.384,-42.707,-179.634,5.512,148.856
C00682=1211.178,2.634,-42.721,-179.631,5.513,148.856
C00683=1211.173,2.903,-42.737,-179.628,5.513,148.855
C00684=1211.166,3.172,-42.753,-179.626,5.514,148.854
C00685=1211.161,3.441,-42.768,-179.623,5.514,148.854
C00686=1211.155,3.710,-42.783,-179.620,5.515,148.853
C00687=1211.150,3.960,-42.797,-179.618,5.515,148.852
C00688=1211.146,4.209,-42.812,-179.615,5.516,148.851
C00689=1211.141,4.458,-42.826,-179.613,5.515,148.851
C00690=1211.136,4.708,-42.841,-179.611,5.516,148.850
C00691=1211.130,4.957,-42.855,-179.608,5.517,148.850
C00692=1211.125,5.207,-42.869,-179.605,5.517,148.849
C00693=1211.120,5.457,-42.883,-179.603,5.518,148.848
C00694=1211.115,5.706,-42.897,-179.600,5.518,148.848
C00695=1211.110,5.956,-42.912,-179.597,5.519,148.847
C00696=1211.106,6.205,-42.927,-179.595,5.519,148.846
C00697=1211.101,6.455,-42.941,-179.593,5.519,148.846
C00698=1211.095,6.704,-42.955,-179.590,5.520,148.845
C00699=1211.090,6.954,-42.969,-179.588,5.520,148.844
C00700=1211.084,7.204,-42.984,-179.585,5.521,148.844
C00701=1211.080,7.453,-42.999,-179.583,5.521,148.843
C00702=1211.075,7.702,-43.013,-179.581,5.521,148.842
C00703=1211.070,7.952,-43.028,-179.578,5.522,148.842
C00704=1211.065,8.202,-43.042,-179.575,5.522,148.841
C00705=1211.060,8.452,-43.056,-179.573,5.523,148.840
C00706=1211.055,8.701,-43.071,-179.570,5.523,148.840
C00707=1211.050,8.950,-43.085,-179.567,5.524,148.839
C00708=1211.045,9.199,-43.099,-179.565,5.525,148.838
C00709=1211.039,9.449,-43.114,-179.563,5.524,148.838
C00710=1211.035,9.698,-43.129,-179.560,5.525,148.837
C00711=1211.030,9.948,-43.143,-179.558,5.525,148.836
C00712=1211.025,10.198,-43.158,-179.555,5.526,148.836
C00713=1211.020,10.447,-43.173,-179.552,5.526,148.835
C00714=1211.015,10.697,-43.187,-179.550,5.527,148.834
C00715=1211.009,10.947,-43.202,-179.547,5.527,148.834
C00716=1211.005,11.196,-43.217,-179.546,5.527,148.833
C00717=1211.000,11.445,-43.231,-179.543,5.528,148.833
C00718=1210.995,11.695,-43.245,-179.540,5.529,148.832
C00719=1210.990,11.944,-43.260,-179.538,5.529,148.831
C00720=1210.984,12.194,-43.275,-179.535,5.530,148.830
C00721=1210.979,12.443,-43.289,-179.532,5.530,148.830
C00722=1210.974,12.692,-43.304,-179.530,5.531,148.829
C00723=1210.969,12.942,-43.318,-179.527,5.531,148.828
C00724=1210.964,13.192,-43.333,-179.525,5.531,148.828
C00725=1210.959,13.441,-43.348,-179.523,5.532,148.827
C00726=1210.954,13.691,-43.363,-179.520,5.532,148.827
C00727=1210.949,13.940,-43.378,-179.518,5.533,148.826
C00728=1210.944,14.190,-43.392,-179.515,5.533,148.825
C00729=1210.939,14.440,-43.407,-179.512,5.534,148.825
C00730=1210.934,14.689,-43.422,-179.510,5.534,148.824
C00731=1210.929,14.939,-43.436,-179.507,5.535,148.823
C00732=1210.924,15.188,-43.451,-179.505,5.535,148.823
C00733=1210.919,15.438,-43.466,-179.503,5.535,148.822
C00734=1210.914,15.687,-43.481,-179.500,5.536,148.821
C00735=1210.909,15.936,-43.495,-179.497,5.536,148.821
C00736=1210.904,16.186,-43.511,-179.495,5.537,148.820
C00737=1210.899,16.436,-43.525,-179.492,5.537,148.819
C00738=1210.894,16.685,-43.540,-179.489,5.538,148.819
C00739=1210.888,16.935,-43.555,-179.487,5.538,148.818
C00740=1210.884,17.184,-43.570,-179.485,5.539,148.817
C00741=1210.879,17.434,-43.584,-179.483,5.539,148.817
C00742=1210.873,17.683,-43.600,-179.480,5.540,148.816
C00743=1210.868,17.933,-43.614,-179.477,5.540,148.815
C00744=1210.864,18.182,-43.629,-179.475,5.541,148.815
C00745=1210.858,18.432,-43.644,-179.472,5.541,148.814
C00746=1210.853,18.681,-43.659,-179.469,5.542,148.813
C00747=1210.849,18.931,-43.674,-179.467,5.543,148.813
C00748=1210.844,19.181,-43.689,-179.465,5.543,148.812
C00749=1210.839,19.430,-43.704,-179.462,5.544,148.812
C00750=1210.834,19.679,-43.718,-179.460,5.543,148.811
C00751=1210.829,19.929,-43.734,-179.457,5.544,148.810
C00752=1210.824,20.179,-43.748,-179.455,5.544,148.810
C00753=1210.818,20.428,-43.764,-179.452,5.545,148.809
C00754=1210.814,20.677,-43.779,-179.449,5.545,148.808
C00755=1210.809,20.927,-43.793,-179.447,5.546,148.808
C00756=1210.803,21.176,-43.809,-179.444,5.547,148.807
C00757=1210.799,21.425,-43.824,-179.442,5.547,148.806
C00758=1210.793,21.675,-43.839,-179.439,5.548,148.806
C00759=1210.788,21.924,-43.854,-179.436,5.548,148.805
C00760=1210.784,22.174,-43.869,-179.434,5.549,148.804
C00761=1210.779,22.424,-43.884,-179.432,5.549,148.804
C00762=1210.774,22.673,-43.899,-179.430,5.549,148.803
C00763=1210.769,22.923,-43.914,-179.427,5.550,148.802
C00764=1210.764,23.172,-43.929,-179.424,5.551,148.802
C00765=1210.758,23.422,-43.944,-179.422,5.551,148.801
C00766=1210.754,23.671,-43.959,-179.419,5.552,148.800
C00767=1210.748,23.920,-43.975,-179.416,5.552,148.800
C00768=1210.743,24.170,-43.989,-179.414,5.553,148.799
C00769=1210.739,24.420,-44.005,-179.412,5.554,148.799
C00770=1210.734,24.669,-44.020,-179.409,5.554,148.798
C00771=1210.729,24.919,-44.036,-179.406,5.555,148.797
C00772=1210.724,25.168,-44.050,-179.404,5.555,148.797
C00773=1210.718,25.418,-44.065,-179.401,5.556,148.796
C00774=1210.714,25.667,-44.080,-179.399,5.555,148.795
C00775=1210.708,25.916,-44.096,-179.397,5.556,148.795
C00776=1210.704,26.166,-44.111,-179.394,5.557,148.794
C00777=1210.698,26.416,-44.126,-179.391,5.557,148.793
C00778=1210.694,26.665,-44.141,-179.389,5.558,148.793
C00779=1210.688,26.915,-44.157,-179.386,5.558,148.792
C00780=1210.684,27.164,-44.172,-179.384,5.559,148.791
C00781=1210.678,27.413,-44.187,-179.381,5.559,148.791
C00782=1210.674,27.663,-44.203,-179.379,5.560,148.790
C00783=1210.669,27.913,-44.218,-179.376,5.561,148.790
C00784=1210.663,28.162,-44.233,-179.373,5.561,148.789
C00785=1210.659,28.411,-44.248,-179.371,5.562,148.788
C00786=1210.653,28.661,-44.264,-179.368,5.562,148.788
C00787=1210.649,28.930,-44.281,-179.366,5.563,148.787
C00788=1210.643,29.199,-44.297,-179.363,5.563,148.786
C00789=1210.638,29.467,-44.314,-179.360,5.564,148.786
C00790=1210.632,29.736,-44.330,-179.358,5.565,148.785
C00791=1210.627,29.985,-44.345,-179.355,5.565,148.784
C00792=1210.622,30.235,-44.361,-179.352,5.566,148.783
C00793=1210.617,30.484,-44.376,-179.350,5.566,148.783
C00794=1210.612,30.734,-44.392,-179.348,5.567,148.782
C00795=1210.607,30.983,-44.407,-179.345,5.568,148.782
C00796=1210.602,31.232,-44.422,-179.342,5.568,148.781
C00797=1210.597,31.482,-44.438,-179.340,5.569,148.780
C00798=1210.592,31.732,-44.454,-179.337,5.569,148.780
C00799=1210.587,31.981,-44.469,-179.335,5.570,148.779
C00800=1210.582,32.230,-44.484,-179.332,5.571,148.779
C00801=1210.577,32.480,-44.500,-179.329,5.571,148.778
C00802=1210.572,32.730,-44.515,-179.327,5.572,148.777
C00803=1210.567,32.979,-44.531,-179.325,5.571,148.776
C00804=1210.562,33.228,-44.547,-179.322,5.572,148.776
C00805=1210.557,33.478,-44.562,-179.320,5.573,148.775
C00806=1210.552,33.728,-44.578,-179.317,5.573,148.775
C00807=1210.547,33.977,-44.593,-179.315,5.574,148.774
C00808=1210.543,34.225,-44.609,-179.312,5.574,148.773
C00809=1210.538,34.476,-44.625,-179.309,5.575,148.773
C00810=1210.532,34.725,-44.640,-179.307,5.575,148.772
C00811=1210.527,34.974,-44.656,-179.305,5.576,148.772
C00812=1210.522,35.223,-44.671,-179.302,5.577,148.771
C00813=1210.518,35.474,-44.687,-179.299,5.577,148.770
C00814=1210.512,35.723,-44.703,-179.297,5.578,148.770
C00815=1210.507,35.972,-44.718,-179.294,5.578,148.769
C00816=1210.503,36.222,-44.733,-179.292,5.579,148.768
C00817=1210.498,36.471,-44.750,-179.289,5.580,148.768
C00818=1210.492,36.720,-44.765,-179.287,5.580,148.767
C00819=1210.487,36.971,-44.781,-179.284,5.581,148.766
C00820=1210.483,37.220,-44.796,-179.281,5.582,148.766
C00821=1210.477,37.469,-44.812,-179.279,5.582,148.765
C00822=1210.473,37.719,-44.828,-179.277,5.583,148.765
C00823=1210.468,37.968,-44.844,-179.274,5.583,148.764
C00824=1210.462,38.217,-44.860,-179.271,5.584,148.763
C00825=1210.458,38.467,-44.875,-179.269,5.585,148.763
C00826=1210.453,38.716,-44.891,-179.266,5.585,148.762
C00827=1210.448,38.965,-44.907,-179.264,5.586,148.761
C00828=1210.443,39.215,-44.923,-179.261,5.587,148.761
C00829=1210.438,39.465,-44.939,-179.259,5.587,148.760
C00830=1210.432,39.714,-44.954,-179.256,5.588,148.759
C00831=1210.428,39.964,-44.971,-179.253,5.588,148.759
C00832=1210.423,40.213,-44.986,-179.251,5.589,148.758
C00833=1210.418,40.463,-45.002,-179.248,5.590,148.758
C00834=1210.413,40.712,-45.017,-179.246,5.590,148.757
C00835=1210.408,40.961,-45.034,-179.243,5.591,148.756
C00836=1210.403,41.211,-45.050,-179.241,5.591,148.756
C00837=1210.398,41.461,-45.065,-179.238,5.592,148.755
C00838=1210.392,41.709,-45.081,-179.236,5.593,148.754
C00839=1210.388,41.959,-45.097,-179.233,5.593,148.754
C00840=1210.383,42.209,-45.112,-179.230,5.594,148.753
C00841=1210.379,42.458,-45.129,-179.228,5.594,148.752
C00842=1210.373,42.707,-45.145,-179.225,5.595,148.752
C00843=1210.368,42.958,-45.161,-179.223,5.596,148.751
C00844=1210.363,43.206,-45.177,-179.220,5.596,148.751
C00845=1210.358,43.456,-45.193,-179.218,5.597,148.750
C00846=1210.353,43.705,-45.209,-179.215,5.597,148.749
C00847=1210.348,43.955,-45.225,-179.212,5.598,148.749
C00848=1210.343,44.205,-45.241,-179.210,5.599,148.748
C00849=1210.338,44.453,-45.257,-179.208,5.599,148.748
C00850=1210.333,44.704,-45.273,-179.205,5.600,148.747
C00851=1210.328,44.952,-45.289,-179.202,5.600,148.746
C00852=1210.323,45.202,-45.305,-179.200,5.601,148.746
C00853=1210.318,45.451,-45.322,-179.198,5.602,148.745
C00854=1210.313,45.701,-45.337,-179.195,5.602,148.744
C00855=1210.309,45.950,-45.354,-179.192,5.603,148.744
C00856=1210.303,46.200,-45.369,-179.190,5.603,148.743
C00857=1210.299,46.449,-45.386,-179.188,5.604,148.743
C00858=1210.293,46.698,-45.402,-179.185,5.605,148.742
C00859=1210.289,46.948,-45.418,-179.182,5.605,148.741
C00860=1210.283,47.197,-45.434,-179.180,5.606,148.741
C00861=1210.279,47.447,-45.451,-179.177,5.607,148.740
C00862=1210.274,47.696,-45.466,-179.175,5.607,148.739
C00863=1210.269,47.946,-45.483,-179.172,5.608,148.739
C00864=1210.264,48.195,-45.498,-179.169,5.609,148.738
C00865=1210.259,48.445,-45.515,-179.166,5.610,148.737
C00866=1210.254,48.694,-45.531,-179.164,5.610,148.737
C00867=1210.249,48.943,-45.547,-179.162,5.611,148.736
C00868=1210.244,49.192,-45.564,-179.159,5.612,148.736
C00869=1210.240,49.442,-45.580,-179.156,5.612,148.735
C00870=1210.234,49.691,-45.596,-179.154,5.613,148.734
C00871=1210.230,49.941,-45.612,-179.152,5.614,148.734
C00872=1210.225,50.190,-45.628,-179.149,5.614,148.733
C00873=1210.219,50.440,-45.645,-179.146,5.615,148.733
C00874=1210.214,50.689,-45.661,-179.144,5.616,148.732
C00875=1210.210,50.939,-45.678,-179.141,5.616,148.731
C00876=1210.205,51.188,-45.694,-179.139,5.617,148.731
C00877=1210.200,51.438,-45.710,-179.136,5.618,148.730
C00878=1210.195,51.687,-45.727,-179.134,5.618,148.729
C00879=1210.190,51.936,-45.743,-179.131,5.619,148.729
C00880=1210.185,52.186,-45.759,-179.129,5.620,148.728
C00881=1210.179,52.435,-45.776,-179.126,5.620,148.728
C00882=1210.175,52.685,-45.792,-179.124,5.621,148.727
C00883=1210.170,52.934,-45.808,-179.121,5.621,148.726
C00884=1210.165,53.183,-45.825,-179.118,5.623,148.726
C00885=1210.161,53.433,-45.841,-179.116,5.623,148.725
C00886=1210.156,53.682,-45.858,-179.113,5.624,148.725
C00887=1210.150,53.932,-45.874,-179.110,5.625,148.724
C00888=1210.145,54.181,-45.891,-179.108,5.625,148.723
C00889=1210.140,54.430,-45.907,-179.105,5.626,148.723
C00890=1210.136,54.680,-45.924,-179.103,5.627,148.722
C00891=1210.130,54.948,-45.941,-179.100,5.627,148.721
C00892=1210.124,55.216,-45.959,-179.098,5.628,148.721
C00893=1210.119,55.486,-45.977,-179.094,5.629,148.720
C00894=1210.114,55.754,-45.994,-179.092,5.630,148.719
C00895=1210.109,56.003,-46.012,-179.089,5.630,148.719
C00896=1210.104,56.252,-46.028,-179.087,5.631,148.718
C00897=1210.099,56.502,-46.044,-179.084,5.632,148.718
C00898=1210.095,56.752,-46.061,-179.082,5.632,148.717
C00899=1210.089,57.001,-46.077,-179.079,5.633,148.716
C00900=1210.084,57.250,-46.094,-179.077,5.634,148.716
C00901=1210.080,57.500,-46.111,-179.074,5.634,148.715
C00902=1210.075,57.749,-46.127,-179.071,5.636,148.715
C00903=1210.070,57.998,-46.144,-179.068,5.636,148.714
C00904=1210.065,58.248,-46.161,-179.066,5.637,148.714
C00905=1210.060,58.497,-46.177,-179.064,5.638,148.713
C00906=1210.055,58.747,-46.194,-179.061,5.638,148.712
C00907=1210.050,58.996,-46.211,-179.058,5.639,148.712
C00908=1210.045,59.245,-46.227,-179.056,5.640,148.711
C00909=1210.040,59.495,-46.243,-179.054,5.640,148.710
C00910=1210.035,59.745,-46.261,-179.051,5.641,148.710
C00911=1210.030,59.993,-46.277,-179.048,5.641,148.709
C00912=1210.026,60.243,-46.294,-179.046,5.642,148.709
C00913=1210.020,60.493,-46.311,-179.043,5.644,148.708
C00914=1210.015,60.741,-46.327,-179.040,5.644,148.707
C00915=1210.010,60.991,-46.345,-179.038,5.645,148.707
C00916=1210.006,61.241,-46.361,-179.036,5.646,148.706
C00917=1210.001,61.489,-46.378,-179.033,5.646,148.706
C00918=1209.995,61.739,-46.395,-179.030,5.647,148.705
C00919=1209.991,61.989,-46.411,-179.028,5.647,148.704
C00920=1209.986,62.238,-46.428,-179.026,5.648,148.704
C00921=1209.981,62.487,-46.445,-179.023,5.649,148.703
C00922=1209.976,62.737,-46.462,-179.020,5.650,148.702
C00923=1209.971,62.987,-46.479,-179.017,5.651,148.702
C00924=1209.966,63.236,-46.496,-179.015,5.652,148.701
C00925=1209.961,63.485,-46.512,-179.012,5.652,148.701
C00926=1209.956,63.734,-46.530,-179.010,5.653,148.700
C00927=1209.952,63.984,-46.547,-179.008,5.654,148.700
C00928=1209.947,64.233,-46.564,-179.005,5.654,148.699
C00929=1209.942,64.482,-46.580,-179.002,5.655,148.698
C00930=1209.936,64.732,-46.597,-179.000,5.655,148.698
C00931=1209.932,64.981,-46.614,-178.997,5.657,148.697
C00932=1209.927,65.231,-46.631,-178.994,5.658,148.697
C00933=1209.922,65.480,-46.648,-178.992,5.658,148.696
C00934=1209.918,65.729,-46.665,-178.989,5.659,148.695
C00935=1209.912,65.979,-46.682,-178.987,5.660,148.695
C00936=1209.908,66.228,-46.699,-178.984,5.660,148.694
C00937=1209.902,66.477,-46.716,-178.982,5.661,148.693
C00938=1209.898,66.727,-46.733,-178.979,5.662,148.693
C00939=1209.892,66.976,-46.750,-178.976,5.663,148.692
C00940=1209.888,67.225,-46.767,-178.974,5.664,148.692
C00941=1209.883,67.475,-46.784,-178.971,5.664,148.691
C00942=1209.878,67.724,-46.801,-178.969,5.665,148.691
C00943=1209.873,67.974,-46.818,-178.966,5.666,148.690
C00944=1209.868,68.223,-46.835,-178.964,5.666,148.689
C00945=1209.863,68.472,-46.853,-178.961,5.667,148.689
C00946=1209.858,68.722,-46.870,-178.958,5.669,148.688
C00947=1209.854,68.972,-46.887,-178.956,5.669,148.688
C00948=1209.848,69.220,-46.904,-178.953,5.670,148.687
C00949=1209.844,69.470,-46.921,-178.951,5.671,148.686
C00950=1209.838,69.719,-46.938,-178.948,5.671,148.686
C00951=1209.834,69.968,-46.956,-178.946,5.672,148.685
C00952=1209.829,70.218,-46.973,-178.943,5.673,148.685
C00953=1209.824,70.468,-46.989,-178.940,5.674,148.684
C00954=1209.820,70.717,-47.007,-178.938,5.675,148.683
C00955=1209.814,70.966,-47.024,-178.935,5.675,148.683
C00956=1209.809,71.215,-47.041,-178.933,5.676,148.682
C00957=1209.804,71.464,-47.059,-178.930,5.677,148.682
C00958=1209.799,71.714,-47.076,-178.928,5.678,148.681
C00959=1209.795,71.964,-47.093,-178.925,5.679,148.681
C00960=1209.790,72.213,-47.111,-178.922,5.679,148.680
C00961=1209.785,72.462,-47.128,-178.920,5.680,148.679
C00962=1209.780,72.711,-47.145,-178.917,5.681,148.679
C00963=1209.774,72.961,-47.162,-178.915,5.682,148.678
C00964=1209.770,73.210,-47.179,-178.912,5.682,148.677
C00965=1209.765,73.459,-47.197,-178.910,5.684,148.677
C00966=1209.760,73.709,-47.214,-178.907,5.684,148.676
C00967=1209.756,73.958,-47.232,-178.904,5.685,148.676
C00968=1209.750,74.208,-47.249,-178.902,5.686,148.675
C00969=1209.746,74.457,-47.267,-178.899,5.686,148.675
C00970=1209.741,74.706,-47.284,-178.897,5.687,148.674
C00971=1209.736,74.956,-47.302,-178.894,5.689,148.674
C00972=1209.731,75.205,-47.319,-178.892,5.689,148.673
C00973=1209.725,75.454,-47.337,-178.889,5.690,148.672
C00974=1209.721,75.703,-47.353,-178.887,5.691,148.672
C00975=1209.716,75.953,-47.371,-178.884,5.691,148.671
C00976=1209.711,76.202,-47.388,-178.881,5.693,148.671
C00977=1209.707,76.451,-47.406,-178.878,5.693,148.670
C00978=1209.701,76.701,-47.423,-178.876,5.694,148.669
C00979=1209.697,76.950,-47.441,-178.874,5.695,148.669
C00980=1209.691,77.200,-47.458,-178.871,5.695,148.668
C00981=1209.687,77.449,-47.476,-178.869,5.696,148.668
C00982=1209.682,77.698,-47.494,-178.866,5.698,148.667
C00983=1209.677,77.948,-47.511,-178.863,5.698,148.666
C00984=1209.672,78.197,-47.529,-178.861,5.699,148.666
C00985=1209.667,78.447,-47.546,-178.858,5.700,148.665
C00986=1209.663,78.696,-47.564,-178.856,5.700,148.665
C00987=1209.658,78.945,-47.582,-178.853,5.702,148.664
C00988=1209.653,79.195,-47.599,-178.850,5.703,148.664
C00989=1209.648,79.444,-47.617,-178.848,5.703,148.663
C00990=1209.643,79.693,-47.635,-178.845,5.704,148.662
C00991=1209.638,79.942,-47.651,-178.843,5.705,148.662
C00992=1209.633,80.192,-47.669,-178.840,5.706,148.661
C00993=1209.628,80.441,-47.687,-178.837,5.707,148.661
C00994=1209.623,80.691,-47.705,-178.835,5.708,148.660
C00995=1209.618,80.959,-47.724,-178.832,5.708,148.659
C00996=1209.613,81.227,-47.744,-178.829,5.710,148.659
C00997=1209.608,81.496,-47.762,-178.827,5.711,148.658
C00998=1209.602,81.764,-47.781,-178.824,5.712,148.658
C00999=1209.597,82.013,-47.799,-178.821,5.712,148.657
C01000=1209.592,82.263,-47.816,-178.818,5.713,148.656
C01001=1209.588,82.512,-47.834,-178.816,5.714,148.656
C01002=1209.583,82.761,-47.852,-178.813,5.715,148.655
C01003=1209.578,83.010,-47.870,-178.810,5.716,148.655
C01004=1209.573,83.260,-47.887,-178.808,5.717,148.654
C01005=1209.568,83.509,-47.905,-178.806,5.717,148.654
C01006=1209.563,83.759,-47.923,-178.804,5.718,148.653
C01007=1209.559,84.008,-47.941,-178.800,5.720,148.653
C01008=1209.554,84.257,-47.959,-178.798,5.720,148.652
C01009=1209.548,84.507,-47.977,-178.796,5.721,148.651
C01010=1209.543,84.756,-47.995,-178.793,5.722,148.651
C01011=1209.539,85.005,-48.013,-178.790,5.723,148.650
C01012=1209.534,85.254,-48.031,-178.788,5.724,148.650
C01013=1209.529,85.503,-48.049,-178.785,5.725,148.649
C01014=1209.524,85.753,-48.067,-178.782,5.725,148.648
C01015=1209.520,86.002,-48.085,-178.780,5.727,148.648
C01016=1209.515,86.251,-48.102,-178.777,5.728,148.647
C01017=1209.510,86.501,-48.120,-178.774,5.728,148.647
C01018=1209.505,86.750,-48.138,-178.772,5.729,148.646
C01019=1209.500,86.999,-48.155,-178.770,5.730,148.646
C01020=1209.495,87.249,-48.173,-178.767,5.732,148.645
C01021=1209.490,87.498,-48.191,-178.764,5.732,148.645
C01022=1209.485,87.747,-48.210,-178.762,5.733,148.644
C01023=1209.481,87.997,-48.228,-178.760,5.734,148.643
C01024=1209.476,88.246,-48.246,-178.756,5.735,148.643
C01025=1209.471,88.496,-48.264,-178.754,5.736,148.642
C01026=1209.466,88.745,-48.282,-178.752,5.736,148.642
C01027=1209.461,88.994,-48.300,-178.749,5.737,148.641
C01028=1209.456,89.243,-48.318,-178.746,5.739,148.641
C01029=1209.451,89.492,-48.336,-178.744,5.739,148.640
C01030=1209.447,89.742,-48.355,-178.741,5.740,148.639
C01031=1209.442,89.991,-48.373,-178.738,5.742,148.639
C01032=1209.437,90.240,-48.391,-178.736,5.742,148.638
C01033=1209.432,90.490,-48.409,-178.734,5.743,148.638
C01034=1209.427,90.739,-48.427,-178.731,5.744,148.637
C01035=1209.422,90.988,-48.444,-178.728,5.745,148.637
C01036=1209.418,91.238,-48.463,-178.726,5.746,148.636
C01037=1209.413,91.487,-48.482,-178.723,5.747,148.636
C01038=1209.408,91.736,-48.500,-178.720,5.747,148.635
C01039=1209.403,91.985,-48.518,-178.718,5.749,148.634
C01040=1209.398,92.234,-48.536,-178.715,5.750,148.634
C01041=1209.393,92.484,-48.554,-178.713,5.751,148.633
C01042=1209.389,92.733,-48.572,-178.710,5.751,148.633
C01043=1209.384,92.983,-48.590,-178.707,5.753,148.632
C01044=1209.378,93.232,-48.609,-178.705,5.754,148.632
C01045=1209.374,93.481,-48.628,-178.702,5.754,148.631
C01046=1209.369,93.730,-48.646,-178.700,5.756,148.631
C01047=1209.364,93.980,-48.664,-178.697,5.756,148.630
C01048=1209.359,94.229,-48.682,-178.695,5.757,148.629
C01049=1209.354,94.478,-48.700,-178.692,5.758,148.629
C01050=1209.349,94.728,-48.719,-178.689,5.759,148.628
C01051=1209.345,94.977,-48.738,-178.687,5.760,148.628
C01052=1209.340,95.226,-48.756,-178.684,5.761,148.627
C01053=1209.335,95.475,-48.774,-178.682,5.763,148.627
C01054=1209.330,95.725,-48.792,-178.679,5.763,148.626
C01055=1209.325,95.974,-48.811,-178.677,5.764,148.625
C01056=1209.320,96.223,-48.829,-178.674,5.766,148.625
C01057=1209.316,96.473,-48.847,-178.671,5.766,148.624
C01058=1209.311,96.722,-48.865,-178.669,5.767,148.624
C01059=1209.306,96.971,-48.885,-178.666,5.768,148.623
C01060=1209.301,97.220,-48.903,-178.663,5.769,148.623
C01061=1209.296,97.470,-48.921,-178.661,5.770,148.622
C01062=1209.291,97.719,-48.940,-178.659,5.771,148.622
C01063=1209.286,97.968,-48.958,-178.656,5.772,148.621
C01064=1209.282,98.218,-48.977,-178.653,5.773,148.621
C01065=1209.277,98.466,-48.995,-178.651,5.774,148.620
C01066=1209.272,98.716,-49.014,-178.648,5.775,148.620
C01067=1209.267,98.965,-49.032,-178.645,5.776,148.619
C01068=1209.263,99.214,-49.051,-178.643,5.777,148.618
C01069=1209.257,99.464,-49.070,-178.640,5.778,148.618
C01070=1209.253,99.712,-49.088,-178.638,5.779,148.617
C01071=1209.248,99.962,-49.107,-178.635,5.780,148.617
C01072=1209.243,100.212,-49.125,-178.633,5.781,148.616
C01073=1209.238,100.460,-49.144,-178.630,5.782,148.616
C01074=1209.234,100.710,-49.162,-178.627,5.783,148.615
C01075=1209.228,100.959,-49.182,-178.625,5.784,148.615
C01076=1209.223,101.208,-49.200,-178.622,5.785,148.614
C01077=1209.219,101.457,-49.219,-178.620,5.786,148.614
C01078=1209.214,101.707,-49.237,-178.617,5.787,148.613
C01079=1209.210,101.956,-49.256,-178.615,5.788,148.613
C01080=1209.204,102.206,-49.275,-178.612,5.789,148.612
C01081=1209.199,102.454,-49.293,-178.609,5.790,148.611
C01082=1209.195,102.704,-49.312,-178.607,5.791,148.611
C01083=1209.190,102.953,-49.331,-178.604,5.792,148.610
C01084=1209.185,103.202,-49.349,-178.602,5.793,148.610
C01085=1209.180,103.452,-49.369,-178.599,5.794,148.609
C01086=1209.175,103.701,-49.387,-178.597,5.795,148.609
C01087=1209.170,103.951,-49.406,-178.594,5.796,148.608
C01088=1209.166,104.200,-49.424,-178.591,5.798,148.608
C01089=1209.161,104.448,-49.443,-178.589,5.798,148.607
C01090=1209.156,104.698,-49.462,-178.586,5.799,148.607
C01091=1209.151,104.947,-49.481,-178.583,5.800,148.606
C01092=1209.147,105.197,-49.500,-178.581,5.801,148.605
C01093=1209.142,105.446,-49.518,-178.578,5.803,148.605
C01094=1209.136,105.695,-49.538,-178.575,5.803,148.604
C01095=1209.132,105.944,-49.556,-178.573,5.804,148.604
C01096=1209.127,106.193,-49.575,-178.570,5.806,148.603
C01097=1209.123,106.443,-49.594,-178.568,5.807,148.603
C01098=1209.117,106.692,-49.613,-178.565,5.807,148.602
C01099=1209.113,106.960,-49.633,-178.563,5.809,148.602
C01100=1209.107,107.229,-49.653,-178.560,5.810,148.601
C01101=1209.101,107.497,-49.674,-178.557,5.811,148.600
C01102=1209.097,107.766,-49.695,-178.554,5.812,148.600
C01103=1209.092,108.015,-49.713,-178.551,5.813,148.599
C01104=1209.087,108.264,-49.733,-178.549,5.814,148.599
C01105=1209.082,108.513,-49.752,-178.546,5.816,148.598
C01106=1209.078,108.762,-49.771,-178.544,5.816,148.598
C01107=1209.073,109.012,-49.789,-178.541,5.817,148.597
C01108=1209.068,109.261,-49.809,-178.538,5.819,148.597
C01109=1209.063,109.510,-49.828,-178.536,5.820,148.596
C01110=1209.059,109.759,-49.847,-178.534,5.820,148.596
C01111=1209.053,110.009,-49.866,-178.531,5.822,148.595
C01112=1209.049,110.258,-49.885,-178.528,5.823,148.595
C01113=1209.044,110.507,-49.904,-178.526,5.824,148.594
C01114=1209.039,110.756,-49.924,-178.523,5.825,148.594
C01115=1209.034,111.005,-49.942,-178.521,5.826,148.593
C01116=1209.029,111.255,-49.961,-178.518,5.827,148.593
C01117=1209.025,111.504,-49.980,-178.515,5.828,148.592
C01118=1209.020,111.753,-50.000,-178.512,5.830,148.591
C01119=1209.014,112.002,-50.019,-178.510,5.831,148.591
C01120=1209.010,112.251,-50.038,-178.508,5.831,148.590
C01121=1209.005,112.500,-50.057,-178.505,5.833,148.590
C01122=1209.000,112.750,-50.077,-178.502,5.834,148.589
C01123=1208.996,113.000,-50.095,-178.500,5.835,148.589
C01124=1208.991,113.249,-50.115,-178.497,5.836,148.588
C01125=1208.986,113.498,-50.134,-178.495,5.837,148.588
C01126=1208.981,113.747,-50.153,-178.492,5.838,148.587
C01127=1208.977,113.996,-50.173,-178.490,5.839,148.587
C01128=1208.971,114.245,-50.192,-178.487,5.840,148.586
C01129=1208.967,114.495,-50.212,-178.484,5.842,148.586
C01130=1208.962,114.743,-50.230,-178.482,5.842,148.585
C01131=1208.957,114.993,-50.250,-178.479,5.844,148.585
C01132=1208.952,115.242,-50.270,-178.476,5.845,148.584
C01133=1208.948,115.491,-50.288,-178.474,5.846,148.584
C01134=1208.943,115.741,-50.308,-178.471,5.847,148.583
C01135=1208.938,115.989,-50.327,-178.469,5.848,148.583
C01136=1208.933,116.239,-50.347,-178.466,5.849,148.582
C01137=1208.928,116.489,-50.367,-178.464,5.850,148.582
C01138=1208.924,116.737,-50.385,-178.460,5.852,148.581
C01139=1208.919,116.987,-50.405,-178.458,5.853,148.581
C01140=1208.914,117.236,-50.424,-178.456,5.853,148.580
C01141=1208.909,117.485,-50.444,-178.453,5.855,148.580
C01142=1208.905,117.734,-50.463,-178.450,5.856,148.579
C01143=1208.899,117.983,-50.482,-178.448,5.857,148.579
C01144=1208.895,118.233,-50.502,-178.445,5.858,148.578
C01145=1208.890,118.482,-50.522,-178.442,5.860,148.578
C01146=1208.885,118.731,-50.542,-178.440,5.860,148.577
C01147=1208.880,118.980,-50.561,-178.438,5.861,148.577
C01148=1208.876,119.230,-50.580,-178.434,5.863,148.576
C01149=1208.871,119.478,-50.600,-178.432,5.864,148.575
C01150=1208.866,119.728,-50.619,-178.430,5.866,148.575
C01151=1208.861,119.977,-50.639,-178.427,5.866,148.574
C01152=1208.856,120.226,-50.659,-178.424,5.868,148.574
C01153=1208.852,120.475,-50.679,-178.422,5.869,148.573
C01154=1208.847,120.725,-50.698,-178.420,5.870,148.573
C01155=1208.842,120.973,-50.717,-178.416,5.871,148.572
C01156=1208.838,121.223,-50.737,-178.414,5.872,148.572
C01157=1208.833,121.472,-50.757,-178.411,5.873,148.571
C01158=1208.828,121.721,-50.776,-178.409,5.874,148.571
C01159=1208.823,121.970,-50.796,-178.406,5.876,148.570
C01160=1208.818,122.220,-50.816,-178.404,5.877,148.570
C01161=1208.813,122.469,-50.835,-178.401,5.878,148.570
C01162=1208.808,122.718,-50.855,-178.398,5.879,148.569
C01163=1208.804,122.967,-50.875,-178.396,5.881,148.569
C01164=1208.799,123.217,-50.895,-178.393,5.881,148.568
C01165=1208.794,123.465,-50.915,-178.391,5.882,148.567
C01166=1208.789,123.715,-50.934,-178.388,5.884,148.567
C01167=1208.784,123.964,-50.954,-178.386,5.885,148.566
C01168=1208.780,124.212,-50.973,-178.383,5.886,148.566
C01169=1208.775,124.462,-50.993,-178.380,5.887,148.565
C01170=1208.771,124.711,-51.013,-178.378,5.889,148.565
C01171=1208.766,124.960,-51.033,-178.375,5.890,148.564
C01172=1208.761,125.209,-51.052,-178.372,5.891,148.564
C01173=1208.756,125.459,-51.072,-178.370,5.892,148.563
C01174=1208.752,125.708,-51.092,-178.367,5.894,148.563
C01175=1208.747,125.957,-51.112,-178.365,5.894,148.562
C01176=1208.743,126.206,-51.132,-178.362,5.896,148.562
C01177=1208.737,126.455,-51.152,-178.359,5.897,148.561
C01178=1208.732,126.705,-51.171,-178.357,5.898,148.561
C01179=1208.727,126.954,-51.192,-178.354,5.899,148.560
C01180=1208.723,127.204,-51.212,-178.351,5.901,148.560
C01181=1208.717,127.452,-51.232,-178.349,5.902,148.559
C01182=1208.713,127.701,-51.252,-178.347,5.902,148.559
C01183=1208.708,127.950,-51.272,-178.344,5.904,148.558
C01184=1208.704,128.200,-51.292,-178.342,5.905,148.558
C01185=1208.699,128.449,-51.312,-178.339,5.907,148.557
C01186=1208.694,128.698,-51.331,-178.336,5.908,148.557
C01187=1208.689,128.947,-51.352,-178.333,5.909,148.556
C01188=1208.685,129.196,-51.371,-178.331,5.910,148.556
C01189=1208.680,129.445,-51.392,-178.328,5.911,148.555
C01190=1208.675,129.695,-51.411,-178.326,5.912,148.555
C01191=1208.671,129.944,-51.432,-178.323,5.914,148.555
C01192=1208.665,130.193,-51.452,-178.321,5.915,148.554
C01193=1208.660,130.442,-51.472,-178.318,5.917,148.554
C01194=1208.656,130.691,-51.492,-178.315,5.917,148.553
C01195=1208.651,130.940,-51.512,-178.313,5.919,148.553
C01196=1208.647,131.189,-51.532,-178.311,5.920,148.552
C01197=1208.642,131.439,-51.552,-178.307,5.921,148.552
C01198=1208.637,131.688,-51.573,-178.305,5.922,148.551
C01199=1208.632,131.936,-51.593,-178.302,5.924,148.551
C01200=1208.627,132.186,-51.613,-178.300,5.925,148.550
C01201=1208.623,132.435,-51.633,-178.297,5.926,148.550
C01202=1208.618,132.684,-51.653,-178.295,5.927,148.549
C01203=1208.613,132.953,-51.675,-178.292,5.929,148.549
C01204=1208.608,133.221,-51.696,-178.289,5.930,148.548
C01205=1208.602,133.490,-51.718,-178.286,5.932,148.548
C01206=1208.597,133.759,-51.741,-178.284,5.933,148.547
C01207=1208.592,134.008,-51.761,-178.281,5.934,148.547
C01208=1208.588,134.257,-51.781,-178.278,5.935,148.546
C01209=1208.583,134.506,-51.801,-178.276,5.937,148.546
C01210=1208.578,134.755,-51.822,-178.273,5.937,148.545
C01211=1208.573,135.004,-51.842,-178.270,5.939,148.545
C01212=1208.569,135.253,-51.862,-178.268,5.941,148.544
C01213=1208.565,135.502,-51.883,-178.265,5.942,148.544
C01214=1208.559,135.752,-51.903,-178.262,5.943,148.543
C01215=1208.555,136.001,-51.923,-178.260,5.944,148.543
C01216=1208.550,136.250,-51.944,-178.257,5.946,148.542
C01217=1208.545,136.499,-51.965,-178.255,5.947,148.542
C01218=1208.541,136.748,-51.985,-178.252,5.948,148.541
C01219=1208.536,136.998,-52.005,-178.250,5.949,148.541
C01220=1208.531,137.247,-52.026,-178.247,5.951,148.540
C01221=1208.526,137.496,-52.046,-178.244,5.952,148.540
C01222=1208.521,137.744,-52.066,-178.242,5.953,148.539
C01223=1208.516,137.994,-52.087,-178.240,5.954,148.539
C01224=1208.512,138.242,-52.107,-178.236,5.956,148.538
C01225=1208.507,138.491,-52.128,-178.234,5.958,148.538
C01226=1208.502,138.741,-52.148,-178.232,5.959,148.538
C01227=1208.497,138.990,-52.168,-178.228,5.960,148.537
C01228=1208.493,139.239,-52.189,-178.226,5.961,148.537
C01229=1208.488,139.488,-52.210,-178.224,5.963,148.536
C01230=1208.483,139.737,-52.230,-178.221,5.963,148.536
C01231=1208.479,139.986,-52.250,-178.218,5.965,148.535
C01232=1208.474,140.236,-52.271,-178.216,5.966,148.535
C01233=1208.469,140.485,-52.292,-178.213,5.968,148.534
C01234=1208.464,140.734,-52.313,-178.210,5.969,148.534
C01235=1208.460,140.983,-52.333,-178.208,5.970,148.533
C01236=1208.454,141.232,-52.354,-178.205,5.972,148.533
C01237=1208.451,141.482,-52.375,-178.203,5.973,148.532
C01238=1208.446,141.731,-52.395,-178.200,5.974,148.532
C01239=1208.441,141.980,-52.416,-178.198,5.975,148.531
C01240=1208.437,142.229,-52.436,-178.195,5.977,148.531
C01241=1208.431,142.478,-52.457,-178.192,5.978,148.530
C01242=1208.427,142.727,-52.478,-178.190,5.979,148.530
C01243=1208.422,142.976,-52.499,-178.187,5.981,148.530
C01244=1208.417,143.225,-52.519,-178.184,5.982,148.529
C01245=1208.412,143.475,-52.540,-178.182,5.984,148.529
C01246=1208.408,143.723,-52.560,-178.179,5.985,148.528
C01247=1208.403,143.972,-52.582,-178.177,5.986,148.528
C01248=1208.398,144.221,-52.603,-178.174,5.988,148.527
C01249=1208.393,144.470,-52.624,-178.172,5.989,148.527
C01250=1208.389,144.719,-52.644,-178.169,5.990,148.526
C01251=1208.384,144.969,-52.665,-178.166,5.991,148.526
C01252=1208.380,145.218,-52.686,-178.164,5.993,148.525
C01253=1208.375,145.467,-52.707,-178.161,5.995,148.525
C01254=1208.370,145.716,-52.728,-178.159,5.995,148.524
C01255=1208.365,145.965,-52.749,-178.156,5.997,148.524
C01256=1208.361,146.214,-52.769,-178.154,5.998,148.524
C01257=1208.356,146.463,-52.790,-178.151,6.000,148.523
C01258=1208.350,146.712,-52.811,-178.148,6.001,148.523
C01259=1208.346,146.961,-52.832,-178.146,6.002,148.522
C01260=1208.342,147.211,-52.853,-178.143,6.004,148.522
C01261=1208.337,147.460,-52.874,-178.140,6.006,148.521
C01262=1208.332,147.709,-52.895,-178.138,6.006,148.521
C01263=1208.327,147.958,-52.916,-178.135,6.008,148.520
C01264=1208.323,148.207,-52.937,-178.133,6.009,148.520
C01265=1208.318,148.456,-52.958,-178.130,6.011,148.520
C01266=1208.314,148.704,-52.979,-178.127,6.012,148.519
C01267=1208.309,148.954,-53.000,-178.125,6.013,148.519
C01268=1208.304,149.203,-53.021,-178.122,6.015,148.518
C01269=1208.299,149.452,-53.041,-178.120,6.016,148.518
C01270=1208.295,149.701,-53.063,-178.117,6.017,148.517
C01271=1208.289,149.950,-53.084,-178.114,6.019,148.517
C01272=1208.285,150.199,-53.105,-178.112,6.020,148.516
C01273=1208.281,150.449,-53.127,-178.109,6.022,148.516
C01274=1208.275,150.698,-53.147,-178.106,6.023,148.515
C01275=1208.271,150.946,-53.169,-178.104,6.024,148.515
C01276=1208.266,151.195,-53.190,-178.101,6.026,148.515
C01277=1208.261,151.445,-53.211,-178.099,6.027,148.514
C01278=1208.257,151.694,-53.233,-178.096,6.029,148.514
C01279=1208.252,151.943,-53.253,-178.093,6.030,148.513
C01280=1208.247,152.192,-53.275,-178.091,6.031,148.513
C01281=1208.242,152.441,-53.296,-178.088,6.033,148.512
C01282=1208.237,152.689,-53.317,-178.085,6.035,148.512
C01283=1208.234,152.939,-53.338,-178.083,6.036,148.512
C01284=1208.229,153.188,-53.360,-178.080,6.037,148.511
C01285=1208.223,153.437,-53.381,-178.077,6.039,148.511
C01286=1208.219,153.686,-53.402,-178.075,6.040,148.510
C01287=1208.215,153.935,-53.423,-178.073,6.042,148.510
C01288=1208.210,154.184,-53.445,-178.070,6.043,148.509
C01289=1208.205,154.433,-53.466,-178.067,6.044,148.509
C01290=1208.200,154.682,-53.487,-178.065,6.046,148.508
C01291=1208.195,154.932,-53.509,-178.062,6.048,148.508
C01292=1208.191,155.180,-53.530,-178.059,6.048,148.507
C01293=1208.186,155.429,-53.551,-178.057,6.050,148.507
C01294=1208.181,155.678,-53.572,-178.055,6.051,148.507
C01295=1208.177,155.927,-53.595,-178.052,6.053,148.506
C01296=1208.172,156.177,-53.615,-178.049,6.054,148.506
C01297=1208.167,156.425,-53.637,-178.047,6.055,148.505
C01298=1208.163,156.675,-53.658,-178.044,6.057,148.505
C01299=1208.158,156.924,-53.680,-178.041,6.059,148.505
C01300=1208.153,157.172,-53.701,-178.039,6.059,148.504
C01301=1208.149,157.422,-53.723,-178.036,6.061,148.504
C01302=1208.144,157.671,-53.744,-178.033,6.063,148.503
C01303=1208.139,157.919,-53.766,-178.031,6.065,148.503
C01304=1208.134,158.169,-53.787,-178.028,6.065,148.502
C01305=1208.129,158.418,-53.809,-178.026,6.067,148.502
C01306=1208.125,158.666,-53.830,-178.023,6.069,148.501
C01307=1208.120,158.936,-53.853,-178.021,6.070,148.501
C01308=1208.114,159.205,-53.877,-178.018,6.071,148.500
C01309=1208.110,159.474,-53.900,-178.015,6.073,148.500
C01310=1208.104,159.743,-53.924,-178.012,6.075,148.500
C01311=1208.100,159.992,-53.945,-178.009,6.077,148.499
C01312=1208.095,160.242,-53.967,-178.006,6.078,148.499
C01313=1208.091,160.490,-53.988,-178.004,6.079,148.498
C01314=1208.087,160.739,-54.010,-178.001,6.081,148.498
C01315=1208.082,160.988,-54.031,-177.999,6.083,148.497
C01316=1208.077,161.236,-54.053,-177.996,6.084,148.497
C01317=1208.072,161.486,-54.074,-177.994,6.085,148.497
C01318=1208.067,161.735,-54.096,-177.991,6.087,148.496
C01319=1208.063,161.984,-54.118,-177.989,6.088,148.496
C01320=1208.058,162.233,-54.140,-177.986,6.090,148.495
C01321=1208.053,162.482,-54.162,-177.983,6.091,148.495
C01322=1208.049,162.731,-54.184,-177.981,6.093,148.495
C01323=1208.044,162.980,-54.205,-177.978,6.094,148.494
C01324=1208.040,163.229,-54.227,-177.975,6.096,148.494
C01325=1208.034,163.479,-54.249,-177.973,6.097,148.493
C01326=1208.029,163.727,-54.271,-177.970,6.098,148.493
C01327=1208.025,163.977,-54.293,-177.968,6.100,148.492
C01328=1208.020,164.225,-54.314,-177.965,6.102,148.492
C01329=1208.016,164.475,-54.336,-177.962,6.104,148.491
C01330=1208.011,164.723,-54.358,-177.960,6.104,148.491
C01331=1208.007,164.973,-54.380,-177.957,6.106,148.491
C01332=1208.002,165.221,-54.402,-177.955,6.108,148.490
C01333=1207.997,165.470,-54.423,-177.952,6.109,148.490
C01334=1207.993,165.719,-54.446,-177.949,6.111,148.489
C01335=1207.988,165.968,-54.467,-177.947,6.112,148.489
C01336=1207.984,166.217,-54.489,-177.944,6.114,148.489
C01337=1207.978,166.466,-54.512,-177.942,6.115,148.488
C01338=1207.974,166.715,-54.534,-177.939,6.117,148.488
C01339=1207.969,166.964,-54.555,-177.936,6.118,148.487
C01340=1207.965,167.213,-54.577,-177.933,6.120,148.487
C01341=1207.960,167.462,-54.599,-177.931,6.121,148.487
C01342=1207.955,167.711,-54.621,-177.929,6.123,148.486
C01343=1207.951,167.960,-54.643,-177.926,6.125,148.486
C01344=1207.946,168.209,-54.666,-177.923,6.125,148.485
C01345=1207.941,168.458,-54.688,-177.921,6.127,148.485
C01346=1207.937,168.707,-54.710,-177.918,6.129,148.484
C01347=1207.932,168.956,-54.731,-177.915,6.131,148.484
C01348=1207.928,169.205,-54.754,-177.913,6.132,148.484
C01349=1207.922,169.454,-54.776,-177.911,6.134,148.483
C01350=1207.918,169.703,-54.798,-177.907,6.135,148.483
C01351=1207.913,169.951,-54.820,-177.905,6.137,148.482
C01352=1207.909,170.201,-54.842,-177.903,6.138,148.482
C01353=1207.903,170.450,-54.865,-177.900,6.140,148.482
C01354=1207.899,170.699,-54.887,-177.897,6.142,148.481
C01355=1207.894,170.948,-54.908,-177.895,6.143,148.481
C01356=1207.890,171.196,-54.931,-177.892,6.145,148.481
C01357=1207.885,171.446,-54.954,-177.889,6.146,148.480
C01358=1207.880,171.695,-54.975,-177.887,6.148,148.480
C01359=1207.876,171.944,-54.997,-177.884,6.149,148.479
C01360=1207.871,172.192,-55.020,-177.881,6.151,148.479
C01361=1207.866,172.442,-55.043,-177.879,6.152,148.479
C01362=1207.862,172.690,-55.064,-177.877,6.154,148.478
C01363=1207.857,172.940,-55.086,-177.874,6.155,148.478
C01364=1207.853,173.189,-55.110,-177.871,6.157,148.477
C01365=1207.848,173.437,-55.131,-177.869,6.158,148.477
C01366=1207.843,173.687,-55.153,-177.866,6.160,148.476
C01367=1207.838,173.935,-55.176,-177.863,6.162,148.476
C01368=1207.834,174.184,-55.198,-177.861,6.164,148.476
C01369=1207.830,174.434,-55.220,-177.858,6.166,148.475
C01370=1207.824,174.682,-55.243,-177.856,6.166,148.475
C01371=1207.820,174.931,-55.265,-177.853,6.168,148.474
C01372=1207.815,175.179,-55.288,-177.850,6.170,148.474
C01373=1207.810,175.429,-55.310,-177.848,6.172,148.474
C01374=1207.806,175.678,-55.333,-177.845,6.173,148.473
C01375=1207.801,175.927,-55.356,-177.843,6.174,148.473
C01376=1207.797,176.176,-55.378,-177.840,6.176,148.473
C01377=1207.793,176.425,-55.400,-177.837,6.178,148.472
C01378=1207.787,176.674,-55.423,-177.834,6.179,148.472
C01379=1207.783,176.922,-55.445,-177.832,6.181,148.471
C01380=1207.778,177.172,-55.468,-177.830,6.182,148.471
C01381=1207.774,177.420,-55.490,-177.827,6.184,148.471
C01382=1207.769,177.670,-55.513,-177.824,6.186,148.470
C01383=1207.765,177.918,-55.536,-177.822,6.188,148.470
C01384=1207.760,178.167,-55.558,-177.819,6.190,148.469
C01385=1207.755,178.416,-55.581,-177.817,6.191,148.469
C01386=1207.751,178.665,-55.603,-177.814,6.192,148.469
C01387=1207.745,178.914,-55.626,-177.811,6.194,148.468
C01388=1207.741,179.163,-55.648,-177.808,6.196,148.468
C01389=1207.736,179.412,-55.671,-177.806,6.197,148.467
C01390=1207.732,179.661,-55.693,-177.804,6.198,148.467
C01391=1207.727,179.910,-55.716,-177.801,6.200,148.467
C01392=1207.723,180.159,-55.739,-177.798,6.202,148.466
C01393=1207.718,180.408,-55.762,-177.796,6.204,148.466
C01394=1207.713,180.656,-55.784,-177.793,6.206,148.466
C01395=1207.709,180.905,-55.808,-177.790,6.207,148.465
C01396=1207.704,181.155,-55.830,-177.788,6.208,148.465
C01397=1207.700,181.404,-55.853,-177.786,6.210,148.465
C01398=1207.694,181.653,-55.875,-177.782,6.212,148.464
C01399=1207.690,181.901,-55.898,-177.780,6.214,148.464
C01400=1207.685,182.150,-55.921,-177.777,6.215,148.463
C01401=1207.681,182.399,-55.944,-177.774,6.217,148.463
C01402=1207.676,182.648,-55.966,-177.772,6.218,148.462
C01403=1207.672,182.897,-55.989,-177.770,6.220,148.462
C01404=1207.667,183.146,-56.013,-177.767,6.222,148.462
C01405=1207.662,183.395,-56.035,-177.764,6.224,148.461
C01406=1207.658,183.643,-56.058,-177.762,6.225,148.461
C01407=1207.653,183.892,-56.081,-177.759,6.227,148.461
C01408=1207.649,184.141,-56.104,-177.757,6.228,148.460
C01409=1207.644,184.390,-56.127,-177.754,6.230,148.460
C01410=1207.639,184.640,-56.150,-177.752,6.232,148.460
C01411=1207.635,184.909,-56.174,-177.749,6.233,148.459
C01412=1207.629,185.179,-56.199,-177.746,6.235,148.459
C01413=1207.624,185.448,-56.225,-177.743,6.237,148.458
C01414=1207.620,185.718,-56.249,-177.740,6.240,148.458
C01415=1207.614,185.967,-56.272,-177.738,6.241,148.458
C01416=1207.609,186.216,-56.295,-177.735,6.242,148.457
C01417=1207.605,186.464,-56.318,-177.732,6.244,148.457
C01418=1207.601,186.713,-56.341,-177.729,6.246,148.456
C01419=1207.596,186.962,-56.364,-177.727,6.248,148.456
C01420=1207.592,187.211,-56.387,-177.724,6.249,148.456
C01421=1207.587,187.459,-56.410,-177.721,6.251,148.455
C01422=1207.582,187.709,-56.434,-177.719,6.252,148.455
C01423=1207.577,187.958,-56.457,-177.717,6.254,148.455
C01424=1207.573,188.206,-56.480,-177.714,6.256,148.454
C01425=1207.569,188.455,-56.503,-177.711,6.258,148.454
C01426=1207.564,188.704,-56.526,-177.709,6.259,148.454
C01427=1207.559,188.953,-56.550,-177.706,6.261,148.453
C01428=1207.555,189.201,-56.572,-177.703,6.263,148.453
C01429=1207.550,189.450,-56.596,-177.701,6.265,148.452
C01430=1207.545,189.699,-56.619,-177.699,6.266,148.452
C01431=1207.541,189.948,-56.642,-177.696,6.268,148.452
C01432=1207.536,190.198,-56.666,-177.693,6.270,148.451
C01433=1207.532,190.446,-56.688,-177.691,6.271,148.451
C01434=1207.527,190.695,-56.712,-177.688,6.273,148.451
C01435=1207.523,190.944,-56.735,-177.685,6.275,148.450
C01436=1207.518,191.193,-56.758,-177.683,6.277,148.450
C01437=1207.513,191.442,-56.782,-177.680,6.279,148.450
C01438=1207.508,191.691,-56.805,-177.677,6.280,148.449
C01439=1207.503,191.940,-56.828,-177.675,6.282,148.449
C01440=1207.499,192.188,-56.851,-177.673,6.283,148.449
C01441=1207.495,192.437,-56.874,-177.670,6.285,148.448
C01442=1207.490,192.686,-56.898,-177.667,6.287,148.448
C01443=1207.485,192.935,-56.922,-177.665,6.289,148.448
C01444=1207.481,193.184,-56.945,-177.662,6.291,148.447
C01445=1207.476,193.433,-56.968,-177.659,6.292,148.447
C01446=1207.471,193.682,-56.992,-177.656,6.294,148.446
C01447=1207.467,193.931,-57.015,-177.654,6.296,148.446
C01448=1207.462,194.179,-57.039,-177.651,6.298,148.446
C01449=1207.458,194.429,-57.063,-177.648,6.299,148.445
C01450=1207.454,194.677,-57.085,-177.646,6.301,148.445
C01451=1207.449,194.926,-57.109,-177.644,6.302,148.444
C01452=1207.445,195.175,-57.133,-177.641,6.304,148.444
C01453=1207.440,195.424,-57.156,-177.638,6.306,148.444
C01454=1207.435,195.673,-57.179,-177.636,6.308,148.443
C01455=1207.430,195.922,-57.203,-177.633,6.309,148.443
C01456=1207.426,196.170,-57.227,-177.631,6.312,148.443
C01457=1207.421,196.419,-57.250,-177.628,6.313,148.443
C01458=1207.417,196.668,-57.274,-177.626,6.315,148.442
C01459=1207.412,196.917,-57.298,-177.623,6.317,148.442
C01460=1207.408,197.166,-57.321,-177.620,6.319,148.442
C01461=1207.403,197.415,-57.344,-177.618,6.321,148.441
C01462=1207.398,197.663,-57.369,-177.615,6.323,148.441
C01463=1207.394,197.912,-57.392,-177.612,6.324,148.441
C01464=1207.389,198.161,-57.415,-177.610,6.326,148.440
C01465=1207.385,198.410,-57.439,-177.607,6.328,148.440
C01466=1207.380,198.659,-57.463,-177.605,6.329,148.440
C01467=1207.376,198.907,-57.487,-177.602,6.331,148.439
C01468=1207.370,199.156,-57.511,-177.600,6.333,148.439
C01469=1207.365,199.405,-57.534,-177.597,6.335,148.438
C01470=1207.361,199.654,-57.558,-177.594,6.336,148.438
C01471=1207.356,199.903,-57.581,-177.592,6.338,148.438
C01472=1207.352,200.151,-57.606,-177.589,6.340,148.437
C01473=1207.348,200.401,-57.629,-177.586,6.342,148.437
C01474=1207.343,200.649,-57.653,-177.584,6.344,148.437
C01475=1207.339,200.898,-57.677,-177.581,6.345,148.436
C01476=1207.334,201.147,-57.701,-177.578,6.347,148.436
C01477=1207.330,201.396,-57.724,-177.576,6.349,148.436
C01478=1207.325,201.645,-57.749,-177.573,6.351,148.435
C01479=1207.320,201.894,-57.772,-177.571,6.353,148.435
C01480=1207.315,202.142,-57.796,-177.568,6.355,148.435
C01481=1207.311,202.390,-57.820,-177.565,6.356,148.434
C01482=1207.306,202.640,-57.844,-177.563,6.358,148.434
C01483=1207.303,202.889,-57.868,-177.560,6.360,148.434
C01484=1207.297,203.138,-57.892,-177.557,6.362,148.433
C01485=1207.293,203.386,-57.916,-177.555,6.364,148.433
C01486=1207.288,203.635,-57.940,-177.552,6.366,148.433
C01487=1207.284,203.884,-57.964,-177.550,6.368,148.433
C01488=1207.279,204.132,-57.988,-177.547,6.370,148.432
C01489=1207.274,204.382,-58.012,-177.545,6.371,148.432
C01490=1207.270,204.631,-58.036,-177.542,6.373,148.432
C01491=1207.266,204.879,-58.060,-177.539,6.375,148.431
C01492=1207.261,205.128,-58.084,-177.537,6.377,148.431
C01493=1207.257,205.377,-58.108,-177.534,6.379,148.430
C01494=1207.251,205.625,-58.132,-177.531,6.381,148.430
C01495=1207.248,205.874,-58.157,-177.529,6.382,148.430
C01496=1207.243,206.123,-58.180,-177.526,6.384,148.429
C01497=1207.238,206.372,-58.205,-177.523,6.386,148.429
C01498=1207.233,206.621,-58.229,-177.521,6.388,148.429
C01499=1207.229,206.869,-58.253,-177.518,6.390,148.428
C01500=1207.224,207.118,-58.276,-177.516,6.392,148.428
C01501=1207.220,207.367,-58.301,-177.513,6.394,148.428
C01502=1207.215,207.616,-58.325,-177.511,6.396,148.428
C01503=1207.211,207.864,-58.349,-177.508,6.397,148.427
C01504=1207.206,208.113,-58.374,-177.505,6.399,148.427
C01505=1207.202,208.363,-58.398,-177.503,6.401,148.427
C01506=1207.197,208.611,-58.422,-177.500,6.403,148.426
C01507=1207.192,208.860,-58.447,-177.497,6.405,148.426
C01508=1207.188,209.108,-58.471,-177.495,6.407,148.426
C01509=1207.183,209.357,-58.495,-177.492,6.408,148.425
C01510=1207.179,209.606,-58.520,-177.489,6.410,148.425
C01511=1207.174,209.855,-58.544,-177.487,6.412,148.425
C01512=1207.169,210.103,-58.568,-177.485,6.414,148.425
C01513=1207.165,210.352,-58.592,-177.482,6.416,148.424
C01514=1207.160,210.602,-58.617,-177.479,6.418,148.424
C01515=1207.156,210.872,-58.643,-177.477,6.420,148.423
C01516=1207.151,211.142,-58.670,-177.474,6.422,148.423
C01517=1207.145,211.412,-58.696,-177.471,6.424,148.423
C01518=1207.141,211.683,-58.723,-177.468,6.426,148.423
C01519=1207.136,211.931,-58.748,-177.466,6.428,148.422
C01520=1207.131,212.180,-58.772,-177.463,6.430,148.422
C01521=1207.128,212.429,-58.797,-177.460,6.432,148.422
C01522=1207.122,212.678,-58.821,-177.458,6.433,148.421
C01523=1207.118,212.926,-58.845,-177.455,6.435,148.421
C01524=1207.113,213.175,-58.870,-177.452,6.437,148.421
C01525=1207.109,213.424,-58.895,-177.450,6.439,148.420
C01526=1207.104,213.673,-58.919,-177.448,6.441,148.420
C01527=1207.100,213.921,-58.943,-177.445,6.443,148.420
C01528=1207.095,214.171,-58.968,-177.442,6.445,148.419
C01529=1207.091,214.419,-58.992,-177.440,6.447,148.419
C01530=1207.085,214.668,-59.017,-177.436,6.449,148.419
C01531=1207.082,214.917,-59.041,-177.434,6.451,148.418
C01532=1207.077,215.166,-59.066,-177.431,6.453,148.418
C01533=1207.073,215.414,-59.091,-177.429,6.455,148.418
C01534=1207.068,215.663,-59.116,-177.426,6.457,148.418
C01535=1207.064,215.911,-59.140,-177.424,6.459,148.417
C01536=1207.059,216.161,-59.165,-177.421,6.461,148.417
C01537=1207.054,216.409,-59.190,-177.418,6.462,148.417
C01538=1207.049,216.658,-59.214,-177.416,6.464,148.416
C01539=1207.045,216.907,-59.240,-177.413,6.466,148.416
C01540=1207.041,217.155,-59.264,-177.411,6.468,148.416
C01541=1207.036,217.404,-59.289,-177.408,6.470,148.416
C01542=1207.031,217.653,-59.313,-177.406,6.472,148.415
C01543=1207.027,217.901,-59.338,-177.403,6.474,148.415
C01544=1207.023,218.150,-59.363,-177.400,6.476,148.415
C01545=1207.018,218.399,-59.387,-177.397,6.478,148.414
C01546=1207.014,218.648,-59.412,-177.395,6.480,148.414
C01547=1207.009,218.896,-59.438,-177.392,6.482,148.414
C01548=1207.004,219.145,-59.462,-177.390,6.484,148.413
C01549=1207.000,219.394,-59.487,-177.387,6.486,148.413
C01550=1206.995,219.642,-59.512,-177.385,6.488,148.413
C01551=1206.991,219.891,-59.537,-177.382,6.490,148.412
C01552=1206.986,220.140,-59.561,-177.379,6.491,148.412
C01553=1206.982,220.389,-59.587,-177.377,6.494,148.412
C01554=1206.978,220.637,-59.611,-177.374,6.495,148.412
C01555=1206.973,220.886,-59.637,-177.372,6.497,148.411
C01556=1206.968,221.135,-59.662,-177.369,6.499,148.411
C01557=1206.964,221.384,-59.687,-177.367,6.501,148.411
C01558=1206.960,221.632,-59.711,-177.364,6.504,148.411
C01559=1206.954,221.881,-59.736,-177.361,6.506,148.410
C01560=1206.950,222.130,-59.762,-177.359,6.508,148.410
C01561=1206.945,222.378,-59.786,-177.356,6.509,148.410
C01562=1206.942,222.627,-59.812,-177.353,6.511,148.409
C01563=1206.936,222.875,-59.836,-177.351,6.513,148.409
C01564=1206.932,223.124,-59.862,-177.348,6.515,148.409
C01565=1206.927,223.373,-59.887,-177.346,6.517,148.409
C01566=1206.923,223.622,-59.912,-177.343,6.519,148.408
C01567=1206.918,223.870,-59.937,-177.341,6.521,148.408
C01568=1206.914,224.119,-59.962,-177.338,6.523,148.408
C01569=1206.910,224.368,-59.987,-177.335,6.526,148.408
C01570=1206.905,224.617,-60.013,-177.333,6.527,148.407
C01571=1206.900,224.866,-60.038,-177.330,6.529,148.407
C01572=1206.896,225.114,-60.063,-177.327,6.531,148.407
C01573=1206.892,225.363,-60.088,-177.325,6.533,148.406
C01574=1206.887,225.611,-60.113,-177.322,6.535,148.406
C01575=1206.883,225.860,-60.139,-177.320,6.537,148.406
C01576=1206.878,226.108,-60.164,-177.317,6.539,148.405
C01577=1206.873,226.358,-60.189,-177.315,6.541,148.405
C01578=1206.869,226.606,-60.214,-177.312,6.544,148.405
C01579=1206.864,226.855,-60.240,-177.309,6.546,148.405
C01580=1206.861,227.104,-60.265,-177.307,6.547,148.404
C01581=1206.856,227.352,-60.290,-177.304,6.550,148.404
C01582=1206.851,227.601,-60.316,-177.302,6.551,148.404
C01583=1206.846,227.849,-60.340,-177.299,6.553,148.404
C01584=1206.842,228.098,-60.366,-177.297,6.555,148.403
C01585=1206.837,228.346,-60.392,-177.294,6.557,148.403
C01586=1206.833,228.596,-60.417,-177.292,6.559,148.403
C01587=1206.829,228.844,-60.442,-177.289,6.562,148.403
C01588=1206.824,229.092,-60.468,-177.286,6.564,148.402
C01589=1206.819,229.341,-60.494,-177.284,6.566,148.402
C01590=1206.815,229.590,-60.519,-177.281,6.568,148.402
C01591=1206.810,229.839,-60.544,-177.278,6.569,148.402
C01592=1206.806,230.088,-60.570,-177.276,6.571,148.401
C01593=1206.801,230.336,-60.595,-177.274,6.573,148.401
C01594=1206.797,230.585,-60.621,-177.271,6.575,148.401
C01595=1206.793,230.833,-60.647,-177.268,6.578,148.400
C01596=1206.787,231.082,-60.671,-177.265,6.580,148.400
C01597=1206.783,231.331,-60.697,-177.263,6.582,148.400
C01598=1206.779,231.580,-60.723,-177.260,6.584,148.400
C01599=1206.774,231.828,-60.748,-177.258,6.586,148.399
C01600=1206.770,232.077,-60.774,-177.256,6.588,148.399
C01601=1206.766,232.325,-60.800,-177.253,6.590,148.399
C01602=1206.761,232.573,-60.825,-177.250,6.592,148.399
C01603=1206.757,232.822,-60.851,-177.247,6.594,148.398
C01604=1206.752,233.071,-60.877,-177.245,6.596,148.398
C01605=1206.748,233.319,-60.902,-177.242,6.598,148.398
C01606=1206.743,233.568,-60.928,-177.240,6.600,148.398
C01607=1206.738,233.817,-60.954,-177.238,6.602,148.398
C01608=1206.734,234.065,-60.979,-177.235,6.604,148.397
C01609=1206.729,234.314,-61.005,-177.232,6.607,148.397
C01610=1206.725,234.563,-61.031,-177.229,6.609,148.397
C01611=1206.721,234.812,-61.057,-177.227,6.611,148.397
C01612=1206.716,235.060,-61.082,-177.224,6.613,148.396
C01613=1206.712,235.309,-61.108,-177.222,6.614,148.396
C01614=1206.707,235.558,-61.134,-177.220,6.617,148.396
C01615=1206.703,235.806,-61.160,-177.216,6.619,148.395
C01616=1206.698,236.055,-61.185,-177.214,6.621,148.395
C01617=1206.694,236.303,-61.211,-177.212,6.623,148.395
C01618=1206.689,236.552,-61.237,-177.209,6.625,148.395
C01619=1206.684,236.823,-61.265,-177.206,6.627,148.394
C01620=1206.680,237.095,-61.293,-177.203,6.630,148.394
C01621=1206.674,237.367,-61.322,-177.201,6.632,148.394
C01622=1206.669,237.637,-61.350,-177.198,6.635,148.394
C01623=1206.665,237.886,-61.376,-177.195,6.636,148.393
C01624=1206.661,238.135,-61.402,-177.193,6.638,148.393
C01625=1206.657,238.384,-61.427,-177.190,6.640,148.393
C01626=1206.651,238.632,-61.453,-177.187,6.643,148.393
C01627=1206.647,238.880,-61.480,-177.185,6.645,148.392
C01628=1206.643,239.129,-61.506,-177.182,6.647,148.392
C01629=1206.638,239.378,-61.532,-177.180,6.649,148.392
C01630=1206.634,239.627,-61.558,-177.177,6.651,148.392
C01631=1206.629,239.875,-61.584,-177.175,6.653,148.392
C01632=1206.625,240.123,-61.610,-177.172,6.656,148.391
C01633=1206.620,240.373,-61.636,-177.169,6.658,148.391
C01634=1206.616,240.621,-61.662,-177.167,6.660,148.391
C01635=1206.612,240.870,-61.688,-177.164,6.662,148.391
C01636=1206.607,241.119,-61.715,-177.162,6.663,148.390
C01637=1206.602,241.367,-61.740,-177.159,6.666,148.390
C01638=1206.598,241.615,-61.766,-177.156,6.668,148.390
C01639=1206.593,241.864,-61.793,-177.154,6.670,148.390
C01640=1206.589,242.112,-61.819,-177.152,6.672,148.389
C01641=1206.585,242.361,-61.845,-177.149,6.674,148.389
C01642=1206.580,242.610,-61.871,-177.146,6.677,148.389
C01643=1206.576,242.858,-61.898,-177.144,6.679,148.389
C01644=1206.571,243.107,-61.924,-177.141,6.681,148.388
C01645=1206.566,243.356,-61.949,-177.139,6.683,148.388
C01646=1206.563,243.604,-61.976,-177.136,6.685,148.388
C01647=1206.558,243.853,-62.002,-177.134,6.688,148.388
C01648=1206.554,244.101,-62.029,-177.131,6.690,148.388
C01649=1206.549,244.350,-62.055,-177.128,6.692,148.387
C01650=1206.545,244.598,-62.082,-177.126,6.694,148.387
C01651=1206.541,244.847,-62.107,-177.123,6.696,148.387
C01652=1206.536,245.096,-62.134,-177.120,6.698,148.387
C01653=1206.532,245.345,-62.160,-177.118,6.701,148.387
C01654=1206.526,245.592,-62.187,-177.116,6.702,148.386
C01655=1206.522,245.841,-62.213,-177.113,6.705,148.386
C01656=1206.518,246.090,-62.240,-177.110,6.707,148.386
C01657=1206.513,246.338,-62.265,-177.108,6.709,148.386
C01658=1206.509,246.587,-62.292,-177.106,6.711,148.386
C01659=1206.505,246.835,-62.319,-177.103,6.713,148.385
C01660=1206.500,247.084,-62.345,-177.100,6.716,148.385
C01661=1206.496,247.332,-62.372,-177.098,6.718,148.385
C01662=1206.491,247.582,-62.398,-177.095,6.720,148.385
C01663=1206.487,247.830,-62.425,-177.093,6.722,148.384
C01664=1206.482,248.078,-62.452,-177.090,6.725,148.384
C01665=1206.478,248.327,-62.477,-177.087,6.727,148.384
C01666=1206.473,248.575,-62.504,-177.085,6.729,148.384
C01667=1206.469,248.824,-62.531,-177.083,6.731,148.384
C01668=1206.465,249.073,-62.557,-177.080,6.734,148.383
C01669=1206.460,249.321,-62.584,-177.077,6.736,148.383
C01670=1206.456,249.569,-62.611,-177.075,6.738,148.383
C01671=1206.451,249.819,-62.637,-177.072,6.739,148.383
C01672=1206.447,250.067,-62.664,-177.069,6.742,148.383
C01673=1206.442,250.315,-62.691,-177.067,6.744,148.382
C01674=1206.438,250.564,-62.718,-177.065,6.746,148.382
C01675=1206.434,250.813,-62.743,-177.062,6.748,148.382
C01676=1206.429,251.061,-62.771,-177.059,6.751,148.382
C01677=1206.424,251.310,-62.798,-177.057,6.753,148.382
C01678=1206.420,251.558,-62.824,-177.054,6.755,148.381
C01679=1206.416,251.806,-62.851,-177.052,6.757,148.381
C01680=1206.411,252.055,-62.877,-177.049,6.760,148.381
C01681=1206.407,252.304,-62.904,-177.047,6.762,148.381
C01682=1206.402,252.552,-62.931,-177.044,6.764,148.380
C01683=1206.397,252.801,-62.958,-177.042,6.766,148.380
C01684=1206.394,253.049,-62.985,-177.039,6.769,148.380
C01685=1206.389,253.297,-63.012,-177.037,6.771,148.380
C01686=1206.384,253.546,-63.039,-177.034,6.773,148.380
C01687=1206.380,253.794,-63.065,-177.031,6.776,148.380
C01688=1206.375,254.043,-63.091,-177.029,6.778,148.379
C01689=1206.371,254.292,-63.119,-177.026,6.780,148.379
C01690=1206.367,254.541,-63.146,-177.024,6.782,148.379
C01691=1206.363,254.789,-63.172,-177.021,6.785,148.379
C01692=1206.358,255.037,-63.199,-177.018,6.787,148.379
C01693=1206.353,255.286,-63.227,-177.016,6.789,148.378
C01694=1206.349,255.534,-63.254,-177.013,6.792,148.378
C01695=1206.345,255.783,-63.280,-177.011,6.793,148.378
C01696=1206.340,256.031,-63.307,-177.008,6.796,148.378
C01697=1206.336,256.280,-63.334,-177.006,6.797,148.378
C01698=1206.331,256.528,-63.361,-177.003,6.800,148.378
C01699=1206.327,256.777,-63.389,-177.000,6.802,148.377
C01700=1206.323,257.025,-63.415,-176.998,6.804,148.377
C01701=1206.318,257.274,-63.442,-176.995,6.807,148.377
C01702=1206.314,257.522,-63.470,-176.993,6.809,148.377
C01703=1206.309,257.770,-63.497,-176.990,6.811,148.376
C01704=1206.305,258.019,-63.524,-176.988,6.814,148.376
C01705=1206.300,258.267,-63.551,-176.985,6.816,148.376
C01706=1206.297,258.516,-63.578,-176.983,6.818,148.376
C01707=1206.292,258.765,-63.605,-176.980,6.820,148.376
C01708=1206.287,259.013,-63.632,-176.978,6.823,148.376
C01709=1206.283,259.262,-63.659,-176.975,6.825,148.375
C01710=1206.278,259.510,-63.687,-176.973,6.827,148.375
C01711=1206.274,259.758,-63.714,-176.970,6.830,148.375
C01712=1206.270,260.007,-63.741,-176.967,6.832,148.375
C01713=1206.265,260.256,-63.768,-176.965,6.834,148.375
C01714=1206.260,260.504,-63.796,-176.962,6.837,148.375
C01715=1206.257,260.752,-63.823,-176.960,6.839,148.374
C01716=1206.252,261.000,-63.850,-176.957,6.841,148.374
C01717=1206.248,261.249,-63.877,-176.955,6.844,148.374
C01718=1206.243,261.498,-63.904,-176.952,6.846,148.374
C01719=1206.239,261.746,-63.932,-176.950,6.848,148.374
C01720=1206.234,261.994,-63.959,-176.947,6.851,148.373
C01721=1206.230,262.244,-63.987,-176.945,6.853,148.373
C01722=1206.226,262.491,-64.014,-176.942,6.855,148.373
C01723=1206.221,262.764,-64.045,-176.939,6.858,148.373
C01724=1206.216,263.037,-64.074,-176.936,6.860,148.373
C01725=1206.211,263.310,-64.104,-176.934,6.863,148.373
C01726=1206.206,263.583,-64.135,-176.931,6.865,148.372
C01727=1206.201,263.831,-64.162,-176.929,6.867,148.372
C01728=1206.197,264.079,-64.189,-176.925,6.870,148.372
C01729=1206.193,264.328,-64.217,-176.923,6.872,148.372
C01730=1206.188,264.576,-64.245,-176.921,6.874,148.372
C01731=1206.184,264.825,-64.272,-176.918,6.877,148.372
C01732=1206.180,265.073,-64.300,-176.916,6.879,148.372
C01733=1206.175,265.322,-64.327,-176.913,6.882,148.371
C01734=1206.171,265.570,-64.355,-176.911,6.884,148.371
C01735=1206.166,265.818,-64.382,-176.908,6.886,148.371
C01736=1206.163,266.067,-64.410,-176.905,6.889,148.371
C01737=1206.158,266.315,-64.437,-176.903,6.891,148.371
C01738=1206.154,266.563,-64.465,-176.900,6.893,148.371
C01739=1206.149,266.813,-64.493,-176.898,6.896,148.371
C01740=1206.144,267.061,-64.521,-176.895,6.898,148.370
C01741=1206.140,267.309,-64.548,-176.893,6.900,148.370
C01742=1206.136,267.558,-64.576,-176.890,6.903,148.370
C01743=1206.131,267.806,-64.603,-176.888,6.905,148.370
C01744=1206.127,268.054,-64.631,-176.885,6.908,148.370
C01745=1206.123,268.303,-64.659,-176.882,6.910,148.369
C01746=1206.118,268.551,-64.686,-176.880,6.912,148.369
C01747=1206.114,268.799,-64.714,-176.877,6.915,148.369
C01748=1206.109,269.049,-64.742,-176.875,6.917,148.369
C01749=1206.105,269.296,-64.769,-176.873,6.919,148.369
C01750=1206.101,269.544,-64.797,-176.870,6.922,148.369
C01751=1206.096,269.794,-64.825,-176.867,6.924,148.369
C01752=1206.092,270.042,-64.853,-176.864,6.927,148.368
C01753=1206.088,270.290,-64.881,-176.862,6.929,148.368
C01754=1206.083,270.539,-64.908,-176.860,6.931,148.368
C01755=1206.078,270.787,-64.937,-176.857,6.934,148.368
C01756=1206.074,271.035,-64.965,-176.855,6.936,148.368
C01757=1206.070,271.283,-64.992,-176.852,6.939,148.368
C01758=1206.066,271.533,-65.020,-176.849,6.941,148.368
C01759=1206.061,271.781,-65.048,-176.847,6.943,148.367
C01760=1206.057,272.029,-65.076,-176.845,6.946,148.367
C01761=1206.053,272.277,-65.104,-176.842,6.948,148.367
C01762=1206.048,272.526,-65.131,-176.839,6.951,148.367
C01763=1206.044,272.775,-65.160,-176.837,6.953,148.367
C01764=1206.039,273.022,-65.188,-176.835,6.955,148.367
C01765=1206.036,273.271,-65.216,-176.832,6.958,148.367
C01766=1206.030,273.519,-65.244,-176.829,6.960,148.366
C01767=1206.026,273.767,-65.272,-176.827,6.963,148.366
C01768=1206.022,274.016,-65.299,-176.824,6.965,148.366
C01769=1206.017,274.264,-65.328,-176.821,6.968,148.366
C01770=1206.013,274.513,-65.356,-176.819,6.970,148.366
C01771=1206.008,274.761,-65.384,-176.817,6.972,148.366
C01772=1206.004,275.010,-65.412,-176.814,6.975,148.366
C01773=1206.000,275.258,-65.440,-176.812,6.977,148.366
C01774=1205.996,275.507,-65.469,-176.809,6.980,148.366
C01775=1205.991,275.754,-65.497,-176.806,6.982,148.365
C01776=1205.987,276.003,-65.525,-176.804,6.985,148.365
C01777=1205.982,276.251,-65.553,-176.801,6.987,148.365
C01778=1205.979,276.500,-65.581,-176.799,6.989,148.365
C01779=1205.974,276.748,-65.610,-176.796,6.992,148.365
C01780=1205.970,276.997,-65.638,-176.794,6.994,148.365
C01781=1205.965,277.245,-65.666,-176.791,6.997,148.365
C01782=1205.961,277.493,-65.694,-176.789,6.999,148.364
C01783=1205.956,277.742,-65.723,-176.786,7.002,148.364
C01784=1205.952,277.990,-65.751,-176.784,7.004,148.364
C01785=1205.948,278.238,-65.779,-176.781,7.006,148.364
C01786=1205.943,278.487,-65.808,-176.779,7.009,148.364
C01787=1205.939,278.735,-65.836,-176.776,7.012,148.364
C01788=1205.934,278.984,-65.864,-176.774,7.015,148.364
C01789=1205.931,279.232,-65.893,-176.771,7.016,148.364
C01790=1205.926,279.480,-65.921,-176.768,7.019,148.364
C01791=1205.922,279.728,-65.949,-176.766,7.022,148.363
C01792=1205.917,279.977,-65.978,-176.763,7.024,148.363
C01793=1205.913,280.225,-66.007,-176.761,7.027,148.363
C01794=1205.908,280.473,-66.034,-176.758,7.030,148.363
C01795=1205.904,280.722,-66.064,-176.756,7.032,148.363
C01796=1205.900,280.970,-66.092,-176.754,7.034,148.363
C01797=1205.895,281.218,-66.120,-176.751,7.037,148.363
C01798=1205.891,281.467,-66.148,-176.749,7.039,148.363
C01799=1205.886,281.715,-66.177,-176.746,7.042,148.363
C01800=1205.882,281.963,-66.206,-176.743,7.044,148.362
C01801=1205.878,282.212,-66.234,-176.741,7.047,148.362
C01802=1205.873,282.460,-66.263,-176.739,7.049,148.362
C01803=1205.870,282.709,-66.291,-176.736,7.052,148.362
C01804=1205.865,282.957,-66.320,-176.733,7.054,148.362
C01805=1205.860,283.205,-66.349,-176.731,7.057,148.362
C01806=1205.857,283.454,-66.377,-176.728,7.059,148.362
C01807=1205.852,283.701,-66.406,-176.726,7.062,148.362
C01808=1205.847,283.950,-66.435,-176.723,7.064,148.361
C01809=1205.844,284.199,-66.463,-176.720,7.067,148.361
C01810=1205.839,284.446,-66.492,-176.718,7.069,148.361
C01811=1205.834,284.695,-66.521,-176.716,7.072,148.361
C01812=1205.831,284.943,-66.549,-176.714,7.074,148.361
C01813=1205.826,285.191,-66.578,-176.710,7.077,148.361
C01814=1205.821,285.440,-66.607,-176.708,7.079,148.361
C01815=1205.818,285.688,-66.635,-176.706,7.082,148.361
C01816=1205.813,285.936,-66.664,-176.703,7.084,148.361
C01817=1205.809,286.185,-66.693,-176.700,7.087,148.361
C01818=1205.804,286.434,-66.722,-176.698,7.089,148.361
C01819=1205.800,286.681,-66.751,-176.695,7.092,148.361
C01820=1205.796,286.930,-66.779,-176.693,7.095,148.360
C01821=1205.791,287.178,-66.809,-176.691,7.098,148.360
C01822=1205.787,287.427,-66.837,-176.688,7.100,148.360
C01823=1205.782,287.674,-66.867,-176.685,7.102,148.360
C01824=1205.778,287.923,-66.895,-176.683,7.105,148.360
